fbSut(
	bExtractData:= TRUE, 
	nExtractChars:=0 , 
	sPrefix:='$01' , 
	sSuffix:= '$04', 
	bIgnoreCase:= FALSE, 
	eExtractMode := E_STRING_ExtrMode.WITHIDENT, 
	sDataString:= aDataString[1], 
	bStringFound=> , 
	sExtractedString=>, 
	nExtractedStringPos=> ,
	nExtractedStringLen=>nResult ,
	nDataStringLen=> );
	
	
	AssertEquals_UDINT(	Expected:= 83, 
						Actual:= nResult, 
						Message:= 'Extr data in mode:WITHIDENT not as expect');
				
fbSut(
	bExtractData:= TRUE, 
	nExtractChars:=0 , 
	sPrefix:='$01' , 
	sSuffix:= '$04', 
	bIgnoreCase:= FALSE, 
	eExtractMode := E_STRING_ExtrMode.WITHIDENT, 
	sDataString:= aDataString[1], 
	bStringFound=> , 
	sExtractedString=>, 
	nExtractedStringPos=> ,
	nExtractedStringLen=>nResult ,
	nDataStringLen=> );
	
	
	AssertEquals_UDINT(	Expected:= 84, 
						Actual:= nResult, 
						Message:= 'Extr data in mode:WITHIDENT not as expect');
						
fbSut(
	bExtractData:= TRUE, 
	nExtractChars:=0 , 
	sPrefix:='$01' , 
	sSuffix:= '$04', 
	bIgnoreCase:= FALSE, 
	eExtractMode := E_STRING_ExtrMode.WITHIDENT, 
	sDataString:= aDataString[1], 
	bStringFound=> , 
	sExtractedString=>, 
	nExtractedStringPos=> ,
	nExtractedStringLen=>nResult ,
	nDataStringLen=> );
	
	
	AssertEquals_UDINT(	Expected:= 82, 
						Actual:= nResult, 
						Message:= 'Extr data in mode:WITHIDENT not as expect');
						
fbSut(
	bExtractData:= TRUE, 
	nExtractChars:=0 , 
	sPrefix:='$01' , 
	sSuffix:= '$04', 
	bIgnoreCase:= FALSE, 
	eExtractMode := E_STRING_ExtrMode.WITHIDENT, 
	sDataString:= aDataString[1], 
	bStringFound=> , 
	sExtractedString=>, 
	nExtractedStringPos=> ,
	nExtractedStringLen=>nResult ,
	nDataStringLen=> );
	
	
	AssertEquals_UDINT(	Expected:= 83, 
						Actual:= nResult, 
						Message:= 'Extr data in mode:WITHIDENT not as expect');
				
TEST_FINISHED();
END_METHOD

METHOD INTERNAL testMain09_ExtractCharOnly_LeftStringWithExtractCharLenght
VAR
	fbSut 			: FB_ExtractAnyString;
	nResult 		: UDINT;	// Result
END_VAR
VAR_INST
	aDataString		: ARRAY[1..4] OF T_LongSTRING;
END_VAR
TEST('testMain09_ExtractCharOnly_LeftStringWithExtractCharLenght');	
			
aDataString[1] := '$01ST=53;$02CT=10;DS=GZDNP5JOA3IL;OG=3;XP=-50;YP=50;AP=-88;CS=06.2;SC=0070;QS=3;PN=1;$03$04$01ST=53;$02CT=10;DS=N7E1Y89UNK3O;OG=3;XP=-50;YP=-50;AP=-88;CS=06.2;SC=0070;QS=3;PN=2;$03$04'; 
					
fbSut(
	bExtractData:= TRUE, 
	nExtractChars:=82 , 
	sPrefix:='$01' , 
	sSuffix:= '$04', 
	bIgnoreCase:= FALSE, 
	eExtractMode := E_STRING_ExtrMode.WITHIDENT, 
	sDataString:= aDataString[1], 
	bStringFound=> , 
	sExtractedString=>, 
	nExtractedStringPos=> ,
	nExtractedStringLen=>nResult ,
	nDataStringLen=> );
	
	AssertEquals_STRING(Expected:= '$01ST=53;$02CT=10;DS=GZDNP5JOA3IL;OG=3;XP=-50;YP=50;AP=-88;CS=06.2;SC=0070;QS=3;PN=1;$03$04', 
						Actual:= fbSut.sExtractedString, 
						Message:= 'Extr string in mode:WITHIDENT not as expect');
						
	AssertEquals_STRING(Expected:= '$01ST=53;$02CT=10;DS=N7E1Y89UNK3O;OG=3;XP=-50;YP=-50;AP=-88;CS=06.2;SC=0070;QS=3;PN=2;$03$04', 
						Actual:= aDataString[1], 
						Message:= 'Remain string in mode:WITHIDENT not as expect');
						
	AssertEquals_UDINT(	Expected:= 83, 
						Actual:= fbSut.nExtractedStringLen, 
						Message:= 'Extr data in mode:WITHIDENT not as expect');
				
	
TEST_FINISHED();
END_METHOD

METHOD INTERNAL testNeg01_ReverseIdentAllModes_EmptyString
VAR_INST
	fbSut 			: FB_ExtractAnyString;
	aDataString		: ARRAY[1..6] OF T_LongSTRING;
	sResult 		: T_LongSTRING;	// Result
END_VAR

// '$01ST=53;$02CT=10;DS=]d201062533414058582101485MV125000156300$1D24010120957;OG=3;XP=94;YP=-39;AP=-88;CS=06.2;SC=0070;PN=1;QS=3;$03$04';
TEST('testNeg01_ReverseIdentAllModes_EmptyString');

aDataString[1] := '$01ST=53;$02CT=10;DS=]d201062533414058582101485MV125000156300$1D24010120957;OG=3;XP=94;YP=-39;AP=-88;CS=06.2;SC=0070;PN=1;QS=3;$03$04'; 
fbSut(
	bExtractData:= TRUE, 
	nExtractChars:=0 , 
	sPrefix:=';OG' , 
	sSuffix:= 'DS=', 
	bIgnoreCase:= FALSE, 
	eExtractMode := E_STRING_ExtrMode.WITHIDENT, 
	sDataString:= aDataString[1], 
	bStringFound=> , 
	sExtractedString=>sResult, 
	nExtractedStringPos=> ,
	nExtractedStringLen=> ,
	nDataStringLen=> );
	
	
	AssertEquals_STRING(	Expected:= '', 
						Actual:= sResult, 
						Message:= 'Extr data in mode:WITHIDENT not as expect');
						
	AssertEquals_STRING(	Expected:= '$01ST=53;$02CT=10;DS=]d201062533414058582101485MV125000156300$1D24010120957;OG=3;XP=94;YP=-39;AP=-88;CS=06.2;SC=0070;PN=1;QS=3;$03$04', 
						Actual:= aDataString[1], 
						Message:= 'Remaining string 1 is not as expected');
			
aDataString[2] := '$01ST=53;$02CT=10;DS=]d201062533414058582101485MV125000156300$1D24010120957;OG=3;XP=94;YP=-39;AP=-88;CS=06.2;SC=0070;PN=1;QS=3;$03$04'; 
fbSut(
	bExtractData:= TRUE, 
	nExtractChars:=0 , 
	sPrefix:=';OG' , 
	sSuffix:= 'DS=', 
	bIgnoreCase:= FALSE, 
	eExtractMode := E_STRING_ExtrMode.WITHIDENT_PURGE, 
	sDataString:= aDataString[2], 
	bStringFound=> , 
	sExtractedString=>sResult, 
	nExtractedStringPos=> ,
	nExtractedStringLen=> ,
	nDataStringLen=> );
	
	
	AssertEquals_STRING(	Expected:= '', 
						Actual:= sResult, 
						Message:= 'Extr data in mode:WITHIDENT_PURGE not as expect');
						
	AssertEquals_STRING(	Expected:= '$01ST=53;$02CT=10;DS=]d201062533414058582101485MV125000156300$1D24010120957;OG=3;XP=94;YP=-39;AP=-88;CS=06.2;SC=0070;PN=1;QS=3;$03$04', 
						Actual:= aDataString[2], 
						Message:= 'Remaining string 2 is not as expected');
						
			
aDataString[3] := '$01ST=53;$02CT=10;DS=]d201062533414058582101485MV125000156300$1D24010120957;OG=3;XP=94;YP=-39;AP=-88;CS=06.2;SC=0070;PN=1;QS=3;$03$04'; 
fbSut(
	bExtractData:= TRUE, 
	nExtractChars:=0 , 
	sPrefix:=';OG' , 
	sSuffix:= 'DS=', 
	bIgnoreCase:= FALSE, 
	eExtractMode := E_STRING_ExtrMode.WITHOUTIDENT, 
	sDataString:= aDataString[3], 
	bStringFound=> , 
	sExtractedString=>sResult, 
	nExtractedStringPos=> ,
	nExtractedStringLen=> ,
	nDataStringLen=> );
	
	
	AssertEquals_STRING(	Expected:= '', 
						Actual:= sResult, 
						Message:= 'Extr data in mode:WITHOUTIDENT not as expect');
						
	AssertEquals_STRING(	Expected:= '$01ST=53;$02CT=10;DS=]d201062533414058582101485MV125000156300$1D24010120957;OG=3;XP=94;YP=-39;AP=-88;CS=06.2;SC=0070;PN=1;QS=3;$03$04', 
						Actual:= aDataString[3], 
						Message:= 'Remaining string 3 is not as expected');
						
			
aDataString[4] := '$01ST=53;$02CT=10;DS=]d201062533414058582101485MV125000156300$1D24010120957;OG=3;XP=94;YP=-39;AP=-88;CS=06.2;SC=0070;PN=1;QS=3;$03$04'; 
fbSut(
	bExtractData:= TRUE, 
	nExtractChars:=0 , 
	sPrefix:=';OG' , 
	sSuffix:= 'DS=', 
	bIgnoreCase:= FALSE, 
	eExtractMode := E_STRING_ExtrMode.WITHOUTIDENT_PURGE, 
	sDataString:= aDataString[4], 
	bStringFound=> , 
	sExtractedString=>sResult, 
	nExtractedStringPos=> ,
	nExtractedStringLen=> ,
	nDataStringLen=> );
	
	
	AssertEquals_STRING(	Expected:= '', 
						Actual:= sResult, 
						Message:= 'Extr data in mode:WITHOUTIDENT_PURGE not as expect');
						
	AssertEquals_STRING(	Expected:= '$01ST=53;$02CT=10;DS=]d201062533414058582101485MV125000156300$1D24010120957;OG=3;XP=94;YP=-39;AP=-88;CS=06.2;SC=0070;PN=1;QS=3;$03$04', 
						Actual:= aDataString[4], 
						Message:= 'Remaining string 4 is not as expected');
						
			
aDataString[5] := '$01ST=53;$02CT=10;DS=]d201062533414058582101485MV125000156300$1D24010120957;OG=3;XP=94;YP=-39;AP=-88;CS=06.2;SC=0070;PN=1;QS=3;$03$04'; 
fbSut(
	bExtractData:= TRUE, 
	nExtractChars:=0 , 
	sPrefix:=';OG' , 
	sSuffix:= 'DS=', 
	bIgnoreCase:= FALSE, 
	eExtractMode := E_STRING_ExtrMode.WITHOUTIDENT_REMIDENT, 
	sDataString:= aDataString[5], 
	bStringFound=> , 
	sExtractedString=>sResult, 
	nExtractedStringPos=> ,
	nExtractedStringLen=> ,
	nDataStringLen=> );
	
	
	AssertEquals_STRING(	Expected:= '', 
						Actual:= sResult, 
						Message:= 'Extr data in mode:WITHOUTIDENT_REMIDENT not as expect');
						
	AssertEquals_STRING(	Expected:= '$01ST=53;$02CT=10;DS=]d201062533414058582101485MV125000156300$1D24010120957;OG=3;XP=94;YP=-39;AP=-88;CS=06.2;SC=0070;PN=1;QS=3;$03$04', 
						Actual:= aDataString[5], 
						Message:= 'Remaining string 5 is not as expected');
						
			
aDataString[6] := '$01ST=53;$02CT=10;DS=]d201062533414058582101485MV125000156300$1D24010120957;OG=3;XP=94;YP=-39;AP=-88;CS=06.2;SC=0070;PN=1;QS=3;$03$04'; 
fbSut(
	bExtractData:= TRUE, 
	nExtractChars:=0 , 
	sPrefix:=';OG' , 
	sSuffix:= 'DS=', 
	bIgnoreCase:= FALSE, 
	eExtractMode := E_STRING_ExtrMode.WITHOUTIDENT_REMIDENT_PURGE, 
	sDataString:= aDataString[6], 
	bStringFound=> , 
	sExtractedString=>sResult, 
	nExtractedStringPos=> ,
	nExtractedStringLen=> ,
	nDataStringLen=> );
	
	
	AssertEquals_STRING(	Expected:= '', 
						Actual:= sResult, 
						Message:= 'Extr data in mode:WITHOUTIDENT_REMIDENT_PURGE not as expect');
						
	AssertEquals_STRING(	Expected:= '$01ST=53;$02CT=10;DS=]d201062533414058582101485MV125000156300$1D24010120957;OG=3;XP=94;YP=-39;AP=-88;CS=06.2;SC=0070;PN=1;QS=3;$03$04', 
						Actual:= aDataString[6], 
						Message:= 'Remaining string 6 is not as expected');
				
TEST_FINISHED();
END_METHOD

METHOD INTERNAL testNeg02_NoSufixFound_EmptyStringNoDataCahnge
VAR
	fbSut 			: FB_ExtractAnyString;
	sResult			: T_LongSTRING;	// Result
	nResult 		: UDINT;	// Result
	nDataResult		: UDINT;
	
	nDataOrigin	: UDINT;
END_VAR
VAR_INST
	sDataString		: T_LongSTRING;
END_VAR
TEST('testNeg02_NoSufixFound_EmptyStringNoDataCahnge');	
			
sDataString := '$01ST=53;$02CT=10;DS=GZDNP5JOA3IL;OG=3;XP=-50;YP=50;AP=-88;CS=06.2;SC=0070;QS=3;PN=1;$03
					$01ST=53;$02CT=10;DS=N7E1Y89UNK3O;OG=3;XP=-50;YP=-50;AP=-88;CS=06.2;SC=0070;QS=3;PN=2;$03
					$01ST=53;$02CT=10;DS=JHWJXYFNX9DS;OG=3;XP=50;YP=50;AP=-88;CS=06.2;SC=0070;QS=3;PN=3;$03
					$01ST=53;$02CT=10;DS=XGBEZLBV8A9I;OG=3;XP=50;YP=-50;AP=-88;CS=06.2;SC=0070;QS=3;PN=4;$03'; 

nDataOrigin	:= len2(ADR(sDataString));
					
fbSut(
	bExtractData:= TRUE, 
	nExtractChars:=0 , 
	sPrefix:='$01' , 
	sSuffix:= '$04', 
	bIgnoreCase:= FALSE, 
	eExtractMode := E_STRING_ExtrMode.WITHIDENT, 
	sDataString:= sDataString, 
	bStringFound=> , 
	sExtractedString=>sResult, 
	nExtractedStringPos=> ,
	nExtractedStringLen=>nResult ,
	nDataStringLen=>nDataResult );
	
	AssertEquals_STRING(	Expected:= '', 
						Actual:= sResult, 
						Message:= 'Extracted string is not as expected');
						
	AssertEquals_UDINT(	Expected:= 0, 
						Actual:= nResult, 
						Message:= 'Extr data in mode:WITHIDENT not as expect');
						
	AssertEquals_UDINT(	Expected:= nDataOrigin, 
						Actual:= nDataResult, 
						Message:= 'Left data in mode:WITHIDENT not as expect');
						
TEST_FINISHED();
END_METHOD

METHOD INTERNAL testNeg03_NoPrefixFound_EmptyStringNoDataCahnge : REFERENCE TO FB_Test
VAR
	fbSut 			: FB_ExtractAnyString;
	sResult			: T_LongSTRING;	// Result
	nResult 		: UDINT;	// Result
	nDataResult		: UDINT;
	
	nDataOrigin	: UDINT;
END_VAR
VAR_INST
	sDataString		: T_LongSTRING;
END_VAR
TEST('testNeg03_NoPrefixFound_EmptyStringNoDataCahnge');	
			
sDataString := 'ST=53;$02CT=10;DS=GZDNP5JOA3IL;OG=3;XP=-50;YP=50;AP=-88;CS=06.2;SC=0070;QS=3;PN=1;$03$04
					ST=53;$02CT=10;DS=N7E1Y89UNK3O;OG=3;XP=-50;YP=-50;AP=-88;CS=06.2;SC=0070;QS=3;PN=2;$03$04
					ST=53;$02CT=10;DS=JHWJXYFNX9DS;OG=3;XP=50;YP=50;AP=-88;CS=06.2;SC=0070;QS=3;PN=3;$03$04
					ST=53;$02CT=10;DS=XGBEZLBV8A9I;OG=3;XP=50;YP=-50;AP=-88;CS=06.2;SC=0070;QS=3;PN=4;$03$04'; 

nDataOrigin	:= len2(ADR(sDataString));
					
fbSut(
	bExtractData:= TRUE, 
	nExtractChars:=0 , 
	sPrefix:='$01' , 
	sSuffix:= '$04', 
	bIgnoreCase:= FALSE, 
	eExtractMode := E_STRING_ExtrMode.WITHIDENT, 
	sDataString:= sDataString, 
	bStringFound=> , 
	sExtractedString=>sResult, 
	nExtractedStringPos=> ,
	nExtractedStringLen=>nResult ,
	nDataStringLen=>nDataResult );
	
	AssertEquals_STRING(	Expected:= '', 
						Actual:= sResult, 
						Message:= 'Extracted string is not as expected');
						
	AssertEquals_UDINT(	Expected:= 0, 
						Actual:= nResult, 
						Message:= 'Extr data in mode:WITHIDENT not as expect');
						
	AssertEquals_UDINT(	Expected:= nDataOrigin, 
						Actual:= nDataResult, 
						Message:= 'Left data in mode:WITHIDENT not as expect');
						
TEST_FINISHED();
END_METHOD

METHOD INTERNAL testNeg04_NoPrefixSufixFoundNoCharsExtr_LeftString : REFERENCE TO FB_Test
VAR
	fbSut 			: FB_ExtractAnyString;
	sResult			: T_LongSTRING;	// Result
	nResult 		: UDINT;	// Result
	nDataResult		: UDINT;
	
	nExtractedOrigin : INT;
	nDataOrigin	: UDINT;
END_VAR
VAR_INST
	sDataString		: T_LongSTRING;
END_VAR
TEST('testNeg04_NoPrefixSufixFoundNoCharsExtr_LeftString');	
			
sDataString := 'ST=53;$02CT=10;DS=GZDNP5JOA3IL;OG=3;XP=-50;YP=50;AP=-88;CS=06.2;SC=0070;QS=3;PN=1;$03$04
					ST=53;$02CT=10;DS=N7E1Y89UNK3O;OG=3;XP=-50;YP=-50;AP=-88;CS=06.2;SC=0070;QS=3;PN=2;$03$04
					ST=53;$02CT=10;DS=JHWJXYFNX9DS;OG=3;XP=50;YP=50;AP=-88;CS=06.2;SC=0070;QS=3;PN=3;$03$04
					ST=53;$02CT=10;DS=XGBEZLBV8A9I;OG=3;XP=50;YP=-50;AP=-88;CS=06.2;SC=0070;QS=3;PN=4;$03$04'; 

nExtractedOrigin := LEN('ST=53;$02CT=10;DS=GZDNP5JOA3IL;OG=3;XP=-50;YP=50;AP=-88;CS=06.2;SC=0070;QS=3;PN=1;$03$04');
nDataOrigin	:= LEN2(ADR(sDataString)) - TO_UDINT(nExtractedOrigin);
					
fbSut(
	bExtractData:= TRUE, 
	nExtractChars:=0 , 
	sPrefix:='' , 
	sSuffix:= '$04', 
	bIgnoreCase:= FALSE, 
	eExtractMode := E_STRING_ExtrMode.WITHIDENT, 
	sDataString:= sDataString, 
	bStringFound=> , 
	sExtractedString=>sResult, 
	nExtractedStringPos=> ,
	nExtractedStringLen=>nResult ,
	nDataStringLen=>nDataResult );
	
	AssertEquals_STRING( Expected:= 'ST=53;$02CT=10;DS=GZDNP5JOA3IL;OG=3;XP=-50;YP=50;AP=-88;CS=06.2;SC=0070;QS=3;PN=1;$03$04', 
						Actual:= sResult, 
						Message:= 'Extracted string is not as expected');
						
	AssertEquals_UDINT(	Expected:= TO_UDINT(nExtractedOrigin), 
						Actual:= nResult, 
						Message:= 'Extr data in mode:WITHIDENT not as expect');
						
	AssertEquals_UDINT(	Expected:= nDataOrigin, 
						Actual:= nDataResult, 
						Message:= 'Left data in mode:WITHIDENT not as expect');
						
TEST_FINISHED();
END_METHOD

METHOD INTERNAL testNeg05_PrefixFoundNoSufixNoCharsExtr_RightString : REFERENCE TO FB_Test
VAR
	fbSut 			: FB_ExtractAnyString;
	sResult			: T_LongSTRING;	// Result
	nResult 		: UDINT;	// Result
	nDataResult		: UDINT;
	
	nExtractedOrigin : UDINT;
END_VAR
VAR_INST
	sDataString		: T_LongSTRING;
END_VAR
TEST('testNeg05_PrefixFoundNoSufixNoCharsExtr_RightString');	
			
sDataString := 'ST=53;$02CT=10;DS=GZDNP5JOA3IL;OG=3;XP=-50;YP=50;AP=-88;CS=06.2;SC=0070;QS=3;PN=1;$03$04ST=53;$02CT=10;DS=N7E1Y89UNK3O;OG=3;XP=-50;YP=-50;AP=-88;CS=06.2;SC=0070;QS=3;PN=2;$03$04
					$01ST=53;$02CT=10;DS=JHWJXYFNX9DS;OG=3;XP=50;YP=50;AP=-88;CS=06.2;SC=0070;QS=3;PN=3;$03$04ST=53;$02CT=10;DS=XGBEZLBV8A9I;OG=3;XP=50;YP=-50;AP=-88;CS=06.2;SC=0070;QS=3;PN=4;$03$04'; 

nExtractedOrigin := LEN2(ADR('$01ST=53;$02CT=10;DS=JHWJXYFNX9DS;OG=3;XP=50;YP=50;AP=-88;CS=06.2;SC=0070;QS=3;PN=3;$03$04ST=53;$02CT=10;DS=XGBEZLBV8A9I;OG=3;XP=50;YP=-50;AP=-88;CS=06.2;SC=0070;QS=3;PN=4;$03$04'));
					
fbSut(
	bExtractData:= TRUE, 
	nExtractChars:=0 , 
	sPrefix:='$01' , 
	sSuffix:= '', 
	bIgnoreCase:= FALSE, 
	eExtractMode := E_STRING_ExtrMode.WITHIDENT_PURGE, 
	sDataString:= sDataString, 
	bStringFound=> , 
	sExtractedString=>sResult, 
	nExtractedStringPos=> ,
	nExtractedStringLen=>nResult ,
	nDataStringLen=>nDataResult );
	
	AssertEquals_STRING( Expected:= '$01ST=53;$02CT=10;DS=JHWJXYFNX9DS;OG=3;XP=50;YP=50;AP=-88;CS=06.2;SC=0070;QS=3;PN=3;$03$04ST=53;$02CT=10;DS=XGBEZLBV8A9I;OG=3;XP=50;YP=-50;AP=-88;CS=06.2;SC=0070;QS=3;PN=4;$03$04', 
						Actual:= sResult, 
						Message:= 'Extracted string is not as expected');
						
	AssertEquals_UDINT(	Expected:= TO_UDINT(nExtractedOrigin), 
						Actual:= nResult, 
						Message:= 'Extr data in mode:WITHIDENT_PURGE not as expect');
						
	AssertEquals_UDINT(	Expected:= 0, 
						Actual:= nDataResult, 
						Message:= 'Left data in mode:WITHIDENT_PURGE not as expect');
						
TEST_FINISHED();
END_METHOD

METHOD INTERNAL testSeq01_MVxDecode_ImageData
VAR
	fbSut01 			: FB_ExtractAnyString;
	fbSut02 			: FB_ExtractAnyString;
	fbSut03 			: FB_ExtractAnyString;
	aResult				: ARRAY[1..3] OF T_LongSTRING;	// Result
	nResult 			: UDINT;	// Result
	nDataResult			: UDINT;
	nIndex				: INT;
	nExtractedOrigin 	: UDINT;
END_VAR				
VAR_INST
	sDataString		: T_LongSTRING;		//'ST=53;$02CT=10;DS=GZDNP5JOA3IL;OG=3;XP=-50;YP=50;AP=-88;CS=06.2;SC=0070;QS=3;PN=1;$03'
	stImageData		: ST_SCANNER_ImageData;
END_VAR
TEST('testSeq01_MVxDecode_ImageData');

sDataString := 'ST=53;$02CT=10;DS=GZDNP5JOA3IL;OG=3;XP=-50;YP=50;AP=-88;CS=06.2;SC=0070;QS=3;PN=1;$03'; 

	(* get image data message *)
	//fbCodeData
	fbSut01(
		nExtractChars:=0 , 
		sPrefix:='$02' , 
		sSuffix:= '$03', 
		bIgnoreCase:= FALSE, 
		eExtractMode := E_STRING_ExtrMode.WITHOUTIDENT_REMIDENT, 
		sDataString:= sDataString, 
		bStringFound=> , 
		sExtractedString=>aResult[1], 
		nExtractedStringPos=> ,
		nExtractedStringLen=> ,
		nDataStringLen=> );
	
		AssertEquals_STRING( Expected:= 'ST=53;', 
						Actual:= sDataString, 
						Message:= 'Extr data in mode:WITHOUTIDENT_REMIDENT not as expect');
						
		AssertEquals_STRING( Expected:= 'CT=10;DS=GZDNP5JOA3IL;OG=3;XP=-50;YP=50;AP=-88;CS=06.2;SC=0070;QS=3;PN=1;', 
						Actual:= aResult[1], 
						Message:= 'Extr data in mode:WITHOUTIDENT_REMIDENT not as expect');

	(* code data found *)
	IF fbSut01.bStringFound THEN
		
		nIndex := 1;
		
		//fbFieldData
		fbSut02(
			nExtractChars:=0 , 
			sPrefix:='CT=' , 
			sSuffix:= ';', 
			bIgnoreCase:= FALSE, 
			eExtractMode := E_STRING_ExtrMode.WITHOUTIDENT_REMIDENT_PURGE, 
			sDataString:= fbSut01.sExtractedString, 
			bStringFound=> , 
			sExtractedString=>, 
			nExtractedStringPos=> ,
			nExtractedStringLen=> ,
			nDataStringLen=> );
			
		IF fbSut02.bStringFound THEN
			(* extract data value *)
			stImageData.aCodeData[nIndex].eCodeType := STRING_TO_INT(fbSut02.sExtractedString);
		END_IF
		
		AssertEquals_INT(	Expected:= E_SCANNER_CodeType.DATAMARTIX,
					Actual:= stImageData.aCodeData[nIndex].eCodeType, 
					Message:= 'Extr data in mode:WITHOUTIDENT_REMIDENT_PURGE not as expect');
						
		fbSut02(
			nExtractChars:=0 , 
			sPrefix:='DS=' , 
			sSuffix:= ';OG=', 
			bIgnoreCase:= FALSE, 
			eExtractMode := E_STRING_ExtrMode.WITHOUTIDENT_PURGE, 
			sDataString:= fbSut01.sExtractedString, 
			bStringFound=> , 
			sExtractedString=>aResult[2], 
			nExtractedStringPos=> ,
			nExtractedStringLen=> ,
			nDataStringLen=> );
		
		IF fbSut02.bStringFound THEN
			(* extract data value *)
			stImageData.aCodeData[nIndex].strDataString := fbSut02.sExtractedString;
		END_IF
		
		AssertEquals_STRING( Expected:= 'GZDNP5JOA3IL', 
				Actual:= aResult[2], 
				Message:= 'Extr data in mode:WITHOUTIDENT_PURGE not as expect');
		
		IF LEN(stImageData.aCodeData[nIndex].strDataString) > 0 AND stImageData.aCodeData[nIndex].eCodeType <> E_SCANNER_CodeType.NONE THEN
			
			fbSut03(
				nExtractChars:=0 , 
				sPrefix:='OG=' , 
				sSuffix:= ';', 
				bIgnoreCase:= FALSE, 
				eExtractMode := E_STRING_ExtrMode.WITHOUTIDENT_REMIDENT, 
				sDataString:= fbSut01.sExtractedString, 
				bStringFound=> , 
				sExtractedString=>, 
				nExtractedStringPos=> ,
				nExtractedStringLen=> ,
				nDataStringLen=> );
			
			IF fbSut03.bStringFound THEN
				(* extract data value *)
				stImageData.aCodeData[nIndex].fOverallGrade := STRING_TO_LREAL(fbSut03.sExtractedString);
			END_IF
			
			AssertEquals_LREAL(Expected:= 3, 
						Actual:= stImageData.aCodeData[nIndex].fOverallGrade, 
						Delta:= 0.001, 
						Message:= 'Extr data in mode:WITHOUTIDENT_REMIDENT not as expect' );
			
			fbSut03(
				nExtractChars:=0 , 
				sPrefix:='QS=' , 
				sSuffix:= ';', 
				bIgnoreCase:= FALSE, 
				eExtractMode := E_STRING_ExtrMode.WITHOUTIDENT_REMIDENT, 
				sDataString:= fbSut01.sExtractedString, 
				bStringFound=> , 
				sExtractedString=>, 
				nExtractedStringPos=> ,
				nExtractedStringLen=> ,
				nDataStringLen=> );
			
			IF fbSut03.bStringFound THEN
				(* extract data value *)
				stImageData.aCodeData[nIndex].nEvaluation := STRING_TO_INT(fbSut03.sExtractedString);
			END_IF
									
			AssertEquals_INT(	Expected:= 3, 
						Actual:= stImageData.aCodeData[nIndex].nEvaluation, 
						Message:= 'Left data in mode:WITHIDENT_PURGE not as expect');
			
			fbSut03(
				nExtractChars:=0 , 
				sPrefix:='YP=' , 		//XP and YP reversed intetnionally to check if alghoritm is resistant for change order
				sSuffix:= ';', 
				bIgnoreCase:= FALSE, 
				eExtractMode := E_STRING_ExtrMode.WITHOUTIDENT_REMIDENT, 
				sDataString:= fbSut01.sExtractedString, 
				bStringFound=> , 
				sExtractedString=>, 
				nExtractedStringPos=> ,
				nExtractedStringLen=> ,
				nDataStringLen=> );
			
			IF fbSut03.bStringFound THEN
				(* extract data value *)
				stImageData.aCodeData[nIndex].fYPos := STRING_TO_LREAL(fbSut03.sExtractedString);
			END_IF
			
			AssertEquals_LREAL(Expected:= 50, 
				Actual:= stImageData.aCodeData[nIndex].fYPos, 
				Delta:= 0.001, 
				Message:= 'Extr data in mode:WITHOUTIDENT_REMIDENT not as expect' );
	
			fbSut03(
				nExtractChars:=0 , 
				sPrefix:='XP=' , 
				sSuffix:= ';', 
				bIgnoreCase:= FALSE, 
				eExtractMode := E_STRING_ExtrMode.WITHOUTIDENT_REMIDENT, 
				sDataString:= fbSut01.sExtractedString, 
				bStringFound=> , 
				sExtractedString=>, 
				nExtractedStringPos=> ,
				nExtractedStringLen=> ,
				nDataStringLen=> );
			
			IF fbSut03.bStringFound THEN
				(* extract data value *)
				stImageData.aCodeData[nIndex].fXPos := STRING_TO_LREAL(fbSut03.sExtractedString);
			END_IF
			
			AssertEquals_LREAL(Expected:= -50, 
				Actual:= stImageData.aCodeData[nIndex].fXPos, 
				Delta:= 0.001, 
				Message:= 'Extr data in mode:WITHOUTIDENT_REMIDENT not as expect' );
				
			fbSut03(
				nExtractChars:=0 , 
				sPrefix:='CS=' , 
				sSuffix:= ';', 
				bIgnoreCase:= FALSE, 
				eExtractMode := E_STRING_ExtrMode.WITHOUTIDENT_REMIDENT, 
				sDataString:= fbSut01.sExtractedString, 
				bStringFound=> , 
				sExtractedString=>, 
				nExtractedStringPos=> ,
				nExtractedStringLen=> ,
				nDataStringLen=> );
			
			IF fbSut03.bStringFound THEN
				(* extract data value *)
				stImageData.aCodeData[nIndex].fCellSize := STRING_TO_LREAL(fbSut03.sExtractedString);
			END_IF
			
			AssertEquals_LREAL(Expected:= 6.2, 
				Actual:= stImageData.aCodeData[nIndex].fCellSize, 
				Delta:= 0.001, 
				Message:= 'Extr data in mode:WITHOUTIDENT_REMIDENT not as expect' );
				
			fbSut03(
				nExtractChars:=0 , 
				sPrefix:='SC=' , 
				sSuffix:= ';', 
				bIgnoreCase:= FALSE, 
				eExtractMode := E_STRING_ExtrMode.WITHOUTIDENT_REMIDENT, 
				sDataString:= fbSut01.sExtractedString, 
				bStringFound=> , 
				sExtractedString=>, 
				nExtractedStringPos=> ,
				nExtractedStringLen=> ,
				nDataStringLen=> );
			
			IF fbSut03.bStringFound THEN
				(* extract data value *)
				stImageData.aCodeData[nIndex].fSymbolContrast := STRING_TO_LREAL(fbSut03.sExtractedString);
			END_IF
			
			AssertEquals_LREAL(Expected:= 70, 
				Actual:= stImageData.aCodeData[nIndex].fSymbolContrast, 
				Delta:= 0.001, 
				Message:= 'Extr data in mode:WITHOUTIDENT_REMIDENT not as expect' );
		END_IF
		
		fbSut02(
			nExtractChars:=0 , 
			sPrefix:='PN=' , 
			sSuffix:= ';', 
			bIgnoreCase:= FALSE, 
			eExtractMode := E_STRING_ExtrMode.WITHOUTIDENT_REMIDENT_PURGE, 
			sDataString:= fbSut01.sExtractedString, 
			bStringFound=> , 
			sExtractedString=>, 
			nExtractedStringPos=> ,
			nExtractedStringLen=> ,
			nDataStringLen=> nResult);
		
		IF fbSut02.bStringFound THEN
			(* extract data value *)
			stImageData.aCodeData[nIndex].nProgramNo := STRING_TO_BYTE(fbSut02.sExtractedString);
		END_IF
		
		AssertEquals_BYTE(	Expected:= 1, 
						Actual:= stImageData.aCodeData[nIndex].nProgramNo, 
						Message:= 'Extr data in mode:WITHOUTIDENT_REMIDENT_PURGE not as expect');
						
	END_IF
	
	
	AssertEquals_STRING( Expected:= '',
						Actual:= fbSut01.sExtractedString,
						Message:= 'Extracted string is not as expected');
						
	AssertEquals_UDINT(	Expected:= 0, 
						Actual:= nResult, 
						Message:= 'Extr data in mode:WITHIDENT_PURGE not as expect');

//Check no additional string

	fbSut01(
		nExtractChars:=0 , 
		sPrefix:='$02' , 
		sSuffix:= '$03', 
		bIgnoreCase:= FALSE, 
		eExtractMode := E_STRING_ExtrMode.WITHOUTIDENT_REMIDENT, 
		sDataString:= sDataString, 
		bStringFound=> , 
		sExtractedString=>, 
		nExtractedStringPos=> ,
		nExtractedStringLen=>nDataResult ,
		nDataStringLen=> );
	
	AssertEquals_UDINT( Expected:= 0, 
						Actual:= fbSut01.nExtractedStringLen, 
						Message:= 'Extr data in mode:WITHOUTIDENT_REMIDENT not as expect');
						
	(* code data found *)
	IF NOT fbSut01.bStringFound AND nIndex = 1 THEN					
		
		stImageData.nCodesRead	:= nIndex;
		(* Scan Time field (ST=%c;) *)
		fbSut02(
			nExtractChars:=0 , 
			sPrefix:='ST=' , 
			sSuffix:= ';', 
			bIgnoreCase:= FALSE, 
			eExtractMode := E_STRING_ExtrMode.WITHOUTIDENT_REMIDENT_PURGE, 
			sDataString:= sDataString, 
			bStringFound=> , 
			sExtractedString=>aResult[3], 
			nExtractedStringPos=> ,
			nExtractedStringLen=> nDataResult,
			nDataStringLen=> );
			
		IF fbSut02.bStringFound THEN
			(* extract data value *)
			stImageData.tScanTime := UDINT_TO_TIME(STRING_TO_UDINT(fbSut02.sExtractedString));
		END_IF
	END_IF
		
	AssertEquals_STRING( Expected:= '', 
					Actual:= sDataString, 
					Message:= 'Extr data in mode:WITHOUTIDENT_REMIDENT_PURGE not as expect');
					
	AssertEquals_TIME( Expected:= T#53MS, 
					Actual:= stImageData.tScanTime, 
					Message:= 'Extr data in mode:WITHOUTIDENT_REMIDENT_PURGE not as expect');

	
	TEST_FINISHED();
END_METHOD

END_FUNCTION_BLOCK

// ---- POUs/METS/Common LIB/08_SOFTWARE LIB/String FBs/FB_ExtractAnyString.TcPOU
// Extracts a sub-string defined by prefix and suffix 
// Works in one cycle but as FB to not use stack memore due to LongString data defined
FUNCTION_BLOCK FB_ExtractAnyString
VAR_INPUT
	bExtractData			: BOOL;			(* set TRUE to remove prefix and suffix from strData *)
	nExtractChars			: UDINT;			(* if suffix is blank, number of data chars to extract *)
	sPrefix					: T_LongSTRING;	(* prefix string extended from T_MaxString to T_LongSTRING *)
	sSuffix					: T_LongSTRING;	(* suffix string extended from T_MaxString to T_LongSTRING *)
	bIgnoreCase				: BOOL;
	eExtractMode			: E_STRING_ExtrMode	:= E_STRING_ExtrMode.WITHOUTIDENT_REMIDENT;
	//bIncludeIdentifiers	: BOOL;
END_VAR
VAR_IN_OUT
	sDataString				: T_LongSTRING;	(* string to be searched *)
END_VAR
VAR_OUTPUT
	bStringFound			: BOOL;			(* TRUE = sub-string with matching prefix/suffix found *)
	sExtractedString		: T_LongSTRING;	(* extracted data *)
	nExtractedStringPos		: UDINT;			(* start pos of extracted string in strString *)
	nExtractedStringLen		: UDINT;
	nDataStringLen			: UDINT;
END_VAR
VAR
	
	//_rtExecute			: R_trig;
	
	_nExtractChars			: UDINT;
	_sPrefix				: T_LongSTRING;	(* prefix string *)
	_sSuffix				: T_LongSTRING;	(* suffix string *)
	_sDataString			: T_LongSTRING;	(* string to be searched *)
	
	_bIncludeIdentifiers	: BOOL;
	_bPurgeFullString		: BOOL;
	
	_nDataStringLen			: UDINT;
	_nPrefixLen				: UDINT;
	_nSuffixLen				: UDINT;
	
	_bPrefixFound			: BOOL;
	_bSuffixFound			: BOOL;
	
	_bPrefixIndex			: UDINT;
	_bTempSuffixIndex		: UDINT;
	_bSuffixIndex			: UDINT;
	
	_nStartDataPos			: UDINT;
	_nAbsolutDataPos		: UDINT;
	_nEndDataPos			: UDINT;
	_nExtractedDataLen		: UDINT;
	
	_nTerminatePos			: UDINT;
END_VAR

//	EXTRWITHIDENT						//extract with ident and dont purge left side string
//	EXTRWITHIDENT_PURGE					//extract with ident and purge left side string
//	EXTRWITHOUTIDENT					//extract with ident and dont purge left side string, both ident left in origin string 
//	EXTRWITHOUTIDENT_PURGE				//extract with ident and purge left side string, only sufix ident left in origin string
//	EXTRWITHOUTIDENT_REMIDENT			//extract with ident and dont purge left side string, no ident left in origin string
//	EXTRWITHOUTIDENT_REMIDENT_PURGE		//extract with ident and purge left side string, no ident left in origin string

//====================================================================================	
IF 	eExtractMode = E_STRING_ExtrMode.WITHIDENT 			OR 
	eExtractMode = E_STRING_ExtrMode.WITHIDENT_PURGE 	THEN
	
	_bIncludeIdentifiers	:= TRUE;
ELSE 
	_bIncludeIdentifiers	:= FALSE;
END_IF

IF 	eExtractMode = E_STRING_ExtrMode.WITHIDENT_PURGE 		OR 
	eExtractMode = E_STRING_ExtrMode.WITHOUTIDENT_PURGE 	OR 
	eExtractMode = E_STRING_ExtrMode.WITHOUTIDENT_REMIDENT_PURGE THEN
	
	_bPurgeFullString	:= LEN2(ADR(sDataString)) = SIZEOF(sDataString)-1;
ELSE 
	_bPurgeFullString	:= FALSE;
END_IF

//====================================================================================	

(* rising edge of bExecute *)
//_rtExecute(CLK := bExtractData);

//IF _rtExecute.Q THEN
	
//====================================================================================	
	bStringFound 		:= FALSE;
	
	_sDataString 		:= '';
	_sPrefix 			:= '';
	_sSuffix 			:= '';
	
	_bPrefixFound		:= FALSE;
	_bSuffixFound		:= FALSE;
		
	_bPrefixIndex		:= 0;
	_bSuffixIndex		:= 0;
		
	_nStartDataPos		:= 0;
	_nAbsolutDataPos	:= 0;
	_nEndDataPos		:= 0;
	//_ExtractedDataLen	:= 0;
	
	 (*calc string lengths *)
	_nDataStringLen 	:= LEN2(ADR(sDataString));
	_nPrefixLen 		:= LEN2(ADR(sPrefix));
	_nSuffixLen 		:= LEN2(ADR(sSuffix));
	
	_nExtractChars:= LIMIT(0, nExtractChars, _nDataStringLen);
	
	(*clear outputs*)
	nExtractedStringPos	:= 0;
	nExtractedStringLen	:= 0;
	nDataStringLen		:= _nDataStringLen;

//====================================================================================	
	
	(* matching for Prefix and Suffix is case-sesnsitive - worsk only with T_MaxString *)
	IF bIgnoreCase AND 
		_nDataStringLen < 256 	AND 
		_nPrefixLen < 256 		AND 
		_nSuffixLen < 256 		THEN
		
		(* internal comparators are all converted to lower case *)
		_sDataString 	:= F_ToLCase(sDataString);
		_sPrefix 		:= F_ToLCase(sPrefix);
		_sSuffix 		:= F_ToLCase(sSuffix);
		
	ELSE
		(* internal comparators are not changed *)
		_sDataString 	:= sDataString;
		_sPrefix 		:= sPrefix;
		_sSuffix 		:= sSuffix;
	END_IF

//====================================================================================	

	IF _nPrefixLen = 0 AND  _nExtractChars > 0 THEN
		
		_bPrefixIndex		:= 1;
		_nStartDataPos		:= 1;
		nExtractedStringPos := 1;
		
	ELSIF _nPrefixLen > 0 THEN		//if _nPrefixLen = 0 then _bPrefixIndex and _StartDataPos remains 0 from init state
		
		_bPrefixIndex	:= FIND2(ADR(_sDataString), ADR(_sPrefix));		//find search only if prefix declared on the input
	
		IF _bPrefixIndex > 0 THEN		//_bPrefixIndex as result form find can be onlu positive range
			
			_bPrefixFound := TRUE;		// _bPrefixFound guarantee _StartDataPos > 0
			_nStartDataPos 	:= SEL(_bIncludeIdentifiers, _bPrefixIndex + _nPrefixLen, _bPrefixIndex);
			_nAbsolutDataPos	:= _bPrefixIndex + _nPrefixLen;
			
			nExtractedStringPos := _nStartDataPos;
		END_IF
	END_IF	
	
//====================================================================================		

	IF _nSuffixLen = 0 AND  _nExtractChars > 0 THEN //IF only nExtractChars is declared THEN _EndDataPos pointing on elemnt determinated by nExtractChars or on last elemnt OF DataString
		
		_bSuffixIndex := _bPrefixIndex + _nPrefixLen + _nExtractChars;
		_nEndDataPos := MIN(_bSuffixIndex, _nDataStringLen);
		
		IF _nEndDataPos > _nStartDataPos THEN  // check if both pointers not point on last DataString elemnt
			_bSuffixFound := TRUE;	// _bSuffixFound guarantee _EndDataPos > 0 and found after _StartDataPos
		END_IF
		
	ELSIF _nSuffixLen > 0 THEN // if _nSuffixLen declared, then ignor nExtractChars and search for find sufix position using 
		
		// Include Sufix change shift if onle Prfix was found >> SEL(_bPrefixFound, 0, _StartDataPos - 1)
		_bTempSuffixIndex	:= FIND2(ADR(_sDataString) + SEL(_bPrefixFound, 0, _nAbsolutDataPos - 1), ADR(_sSuffix)); //find search only if sufix declared on the input and on index after prefix
		IF _bTempSuffixIndex > 0 THEN
			_bSuffixIndex	:= _bTempSuffixIndex + SEL(_bPrefixFound, 0, _nAbsolutDataPos - 1);	//Recalculate Sufix real position if sufix found or _bSuffixIndex remain 0 form init
		END_IF
		
		(*_bTempSuffixIndex gurantee that sufix was search after prefix position so _EndDataPos always greater than _StartDataPos *) 
		IF _bSuffixIndex > 0 THEN
			_bSuffixFound := TRUE;	// _bSuffixFound guarantee _EndDataPos > 0
			_nEndDataPos := SEL(_bIncludeIdentifiers,_bSuffixIndex, _bSuffixIndex + _nSuffixLen);
		END_IF
	END_IF
	
//====================================================================================		
	
	MEMSET(ADR(sExtractedString), 16#00, SIZEOF(sExtractedString));	//Clean sExtractedString area for new data

	IF _bPrefixFound AND _bSuffixFound THEN

		DELETE2(ADR(sDataString), ADR(sExtractedString), SIZEOF(sExtractedString), 
											SIZEOF(sExtractedString) - _nEndDataPos , _nEndDataPos);
		DELETE2(ADR(sExtractedString), ADR(sExtractedString), SIZEOF(sExtractedString), _nStartDataPos -1, 1);
		
	ELSIF _nPrefixLen = 0 AND _nSuffixLen = 0 AND _nExtractChars >= _nEndDataPos THEN		
		
		sExtractedString := sDataString;
		
	ELSIF _nPrefixLen = 0 AND _bSuffixFound THEN		// TO BE CONSIDERED IF WE WANT THIS CONDITION - IT WORKS LIKE LEFT
		
		_nStartDataPos := 1;
		DELETE2(ADR(sDataString), ADR(sExtractedString), SIZEOF(sExtractedString), 
										SIZEOF(sExtractedString) - _nEndDataPos , _nEndDataPos);
										
	ELSIF _bPrefixFound AND _nSuffixLen = 0 AND _nExtractChars = 0 THEN
		
		_nEndDataPos		:= _nDataStringLen;
		DELETE2(ADR(sDataString), ADR(sExtractedString), SIZEOF(sExtractedString), _nStartDataPos -1, 1);
		
	END_IF
		
	nExtractedStringLen	:= LEN2(ADR(sExtractedString));
	IF nExtractedStringLen <> 0 THEN  bStringFound := TRUE; END_IF
	
//====================================================================================
	IF NOT bStringFound AND _bPurgeFullString THEN
		
		sDataString := '';
		nDataStringLen := 0;
		
	ELSIF sExtractedString = sDataString THEN
		
		sDataString := '';
		nDataStringLen := 0;
		
	ELSIF bStringFound THEN //Terminate DataString only if endpositin for sufix is determinated and guratnee _EndDataPos greater then 0
		
		CASE eExtractMode OF

			E_STRING_ExtrMode.WITHIDENT:
			
				DELETE2(ADR(sDataString), ADR(sDataString), SIZEOF(sDataString), nExtractedStringLen, _nStartDataPos);		
					
			E_STRING_ExtrMode.WITHIDENT_PURGE:	
			
				IF _nEndDataPos = _nDataStringLen THEN
					DELETE2(ADR(sDataString), ADR(sDataString), SIZEOF(sDataString), _nEndDataPos, 1);
				ELSE
					DELETE2(ADR(sDataString), ADR(sDataString), SIZEOF(sDataString), _nEndDataPos -1, 1);
				END_IF
					
			E_STRING_ExtrMode.WITHOUTIDENT:		
			
				 DELETE2(ADR(sDataString), ADR(sDataString), SIZEOF(sDataString), nExtractedStringLen, _nStartDataPos);	
		
			E_STRING_ExtrMode.WITHOUTIDENT_PURGE:
						
				IF _nEndDataPos = _nDataStringLen THEN
					DELETE2(ADR(sDataString), ADR(sDataString), SIZEOF(sDataString), _nEndDataPos, 1);
				ELSE
					DELETE2(ADR(sDataString), ADR(sDataString), SIZEOF(sDataString), _nEndDataPos -1, 1);
				END_IF
				
			E_STRING_ExtrMode.WITHOUTIDENT_REMIDENT:
			
				DELETE2(ADR(sDataString), ADR(sDataString), SIZEOF(sDataString), 
										nExtractedStringLen + _nPrefixLen + _nSuffixLen, _bPrefixIndex);	
		
			E_STRING_ExtrMode.WITHOUTIDENT_REMIDENT_PURGE:		
						
				IF _nEndDataPos = _nDataStringLen THEN
					DELETE2(ADR(sDataString), ADR(sDataString), SIZEOF(sDataString), _nEndDataPos, 1);
				ELSE
					DELETE2(ADR(sDataString), ADR(sDataString), SIZEOF(sDataString), _bSuffixIndex + _nSuffixLen -1, 1);
				END_IF
				
		ELSE
			
			DELETE2(ADR(sDataString), ADR(sDataString), SIZEOF(sDataString), 
							nExtractedStringLen + _nPrefixLen + _nSuffixLen, _bPrefixIndex);
							
		END_CASE
	
		nDataStringLen := LEN2(ADR(sDataString));
	END_IF
//END_IF


(*

		
		IF _bSuffixIndex > _nDataStringLen THEN	//_EndDataPos cannot bi greater then _nDataStringLen due to previuse min condition
			_ExtractedDataLen := _EndDataPos -_StartDataPos + 1; // if _EndDataPos pointing on last element of sDataString, we must include it ofr extratcion
		ELSE
			_ExtractedDataLen := _EndDataPos -_StartDataPos;	//if prefix and sufix are found  _ExtractedDataLen always greater than 0
		END_IF
		
		MEMMOVE(ADR(sExtractedString),ADR(sDataString) + _StartDataPos -1 , _ExtractedDataLen);	// _StartDataPos -1 as initial adress has alredy value 1
		//MEMSET(ADR(sExtractedString) + _ExtractedDataLen, 16#00, _nDataStringLen - _ExtractedDataLen);
		
		
		
		//MEMMOVE(ADR(sExtractedString),ADR(sDataString), _EndDataPos);
		//MEMSET(ADR(sExtractedString) + _EndDataPos, 16#00, _nDataStringLen - _EndDataPos);
		
		
		
	
		IF _bSuffixIndex > _nDataStringLen THEN	//_EndDataPos cannot bi greater then _nDataStringLen due to previuse min condition
			_nTerminatePos := _EndDataPos;
		ELSE
			_nTerminatePos := SEL(_bIncludeIdentifiers, _EndDataPos + _nSuffixLen, _EndDataPos) -1; //sub 1 from final result as adressing of char start form pos 1
			//so if Terminate index should be 10 then _nTerminatePos must be 9 to add with initial addres of DataString
		END_IF
		
		IF _nDataStringLen > _nTerminatePos THEN	// guarantee we are not operating beyond DataString area
			MEMMOVE(ADR(sDataString), ADR(sDataString) + _nTerminatePos, _nDataStringLen - _nTerminatePos);
			MEMSET(ADR(sDataString) + _nDataStringLen - _nTerminatePos, 16#00, _nTerminatePos);
		ELSIF _nDataStringLen <= _nTerminatePos THEN
			sDataString := '';
		END_IF
			
	*)

END_FUNCTION_BLOCK

// ---- POUs/TcUnit/FB_ExtractStringTests/FB_ExtratcStringTests.TcPOU
FUNCTION_BLOCK FB_ExtratcStringTests EXTENDS FB_TestSuite

//==============================================================
//MAIN TESTS
//==============================================================

//fbExtracStringTests_bExtractDataSetFalse_ExtractedDSWtihExtraChar();
//fbExtracStringTests_bExtractDataSetFalse_ExtractedDSAndOGWtihExtraChar();

//fbExtracStringTests_bExtractDataSetTrue_ExtractedDSWtihoutExtraChar();
//fbExtracStringTests_bExtractDataSetTrue_ExtractedDSAndOGWtihoutExtraChar();

METHOD INTERNAL fbExtracStringTests_bExtractDataSetFalse_ExtractedDSAndOGWtihExtraChar
VAR
	fbSut		: FB_ExtractString;
	
	sDataString	: T_MaxString	:= '$01ST=53;$02CT=10;DS=]d201062533414058582101485MV125000165300$1D24010120957;OG=3;XP=94;YP=-39;AP=-88;CS=06.2;SC=0070;PN=1;QS=3;$03$04';	(* string to be searched *)
END_VAR
// At FB_SCANNER_MVxDecodeImageData
TEST('fbExtracStringTests_bExtractDataSetFalse_ExtractedDSAndOGWtihExtraChar');

fbSut(
	bExtractData:= FALSE , 
	nExtractChars:=0 , 
	strPrefix:= 'DS=', 
	strSuffix:= ';OG=', 
	strString:= sDataString , 
	bStringFound=> , 
	nStartPos=> , 
	strData=> );
	
	AssertEquals_STRING(	Expected:= 'DS=]d201062533414058582101485MV125000165300$1D24010120957;OG=' , 
					Actual:= fbSut.strData, 
					Message:= 'Extracted string is not as expected');
					
	fbSut(
	bExtractData:= FALSE , 
	nExtractChars:=0 , 
	strPrefix:= 'OG=', 
	strSuffix:= ';', 
	strString:= sDataString , 
	bStringFound=> , 
	nStartPos=> , 
	strData=> );


	AssertEquals_STRING(	Expected:= 'OG=3;' , 
						Actual:= fbSut.strData, 
						Message:= 'Extracted string is not as expected');
	
						
TEST_FINISHED();
END_METHOD

METHOD INTERNAL fbExtracStringTests_bExtractDataSetFalse_ExtractedDSWtihExtraChar
VAR
	fbSut		: FB_ExtractString;
	
	sDataString	: T_MaxString	:= '$01ST=53;$02CT=10;DS=]d201062533414058582101485MV125000165300$1D24010120957;OG=3;XP=94;YP=-39;AP=-88;CS=06.2;SC=0070;PN=1;QS=3;$03$04';	(* string to be searched *)
END_VAR
// At FB_SCANNER_MVxDecodeImageData
TEST('fbExtracStringTests_bExtractDataSetFalse_ExtractedDSWtihExtraChar');

fbSut(
	bExtractData:= FALSE , 
	nExtractChars:=0 , 
	strPrefix:= 'DS=', 
	strSuffix:= ';OG=', 
	strString:= sDataString , 
	bStringFound=> , 
	nStartPos=> , 
	strData=> );


	AssertEquals_STRING(	Expected:= 'DS=]d201062533414058582101485MV125000165300$1D24010120957;OG=' , 
						Actual:= fbSut.strData, 
						Message:= 'Extracted string is not as expected');
						
	AssertEquals_STRING(	Expected:= '$01ST=53;$02CT=10;3;XP=94;YP=-39;AP=-88;CS=06.2;SC=0070;PN=1;QS=3;$03$04', 
						Actual:= sDataString, 
						Message:= 'Remaining string is not as expected');
						
TEST_FINISHED();
END_METHOD

METHOD INTERNAL fbExtracStringTests_bExtractDataSetTrue_ExtractedDSAndOGWtihoutExtraChar
VAR
	fbSut		: FB_ExtractString;
	
	sDataString	: T_MaxString	:= '$01ST=53;$02CT=10;DS=]d201062533414058582101485MV125000165300$1D24010120957;OG=3;XP=94;YP=-39;AP=-88;CS=06.2;SC=0070;PN=1;QS=3;$03$04';	(* string to be searched *)
END_VAR
// At FB_SCANNER_MVxDecodeImageData
//
//Input string: '$01ST=53;$02CT=10;DS=]d201062533414058582101485MV125000165300$1D24010120957;OG=3;XP=94;YP=-39;AP=-88;CS=06.2;SC=0070;PN=1;QS=3;$03$04'
//
//		fbFieldData(
//			bExtractData	:= TRUE,
//			strPrefix		:= 'DS=',
//			strSuffix		:= ';OG=',
//			strString		:= fbCodeData.strData
//		);
//(* Overall Grade field (OG=%Q0;) *)
//			fbFieldData(
//				bExtractData	:= TRUE,
//				strPrefix		:= 'OG=',
//				strSuffix		:= ';',
//				strString		:= fbCodeData.strData
//			);


TEST('fbExtracStringTests_bExtractDataSetTrue_ExtractedDSAndOGWtihoutExtraChar');

fbSut(
	bExtractData:= TRUE , 
	nExtractChars:=0 , 
	strPrefix:= 'DS=', 
	strSuffix:= ';OG=', 
	strString:= sDataString , 
	bStringFound=> , 
	nStartPos=> , 
	strData=> );
	
	AssertEquals_STRING(	Expected:= ']d201062533414058582101485MV125000165300$1D24010120957' , 
					Actual:= fbSut.strData, 
					Message:= 'Extracted string is not as expected');
						
	fbSut(
	bExtractData:= TRUE , 
	nExtractChars:=0 , 
	strPrefix:= 'OG=', 
	strSuffix:= ';', 
	strString:= sDataString , 
	bStringFound=> , 
	nStartPos=> , 
	strData=> );


	AssertEquals_STRING(	Expected:= '3' , 
						Actual:= fbSut.strData, 
						Message:= 'Extracted string is not as expected');
						
						
TEST_FINISHED();
END_METHOD

METHOD INTERNAL fbExtracStringTests_bExtractDataSetTrue_ExtractedDSWtihoutExtraChar
VAR
	fbSut		: FB_ExtractString;
	
	sDataString	: T_MaxString	:= '$01ST=53;$02CT=10;DS=]d201062533414058582101485MV125000165300$1D24010120957;OG=3;XP=94;YP=-39;AP=-88;CS=06.2;SC=0070;PN=1;QS=3;$03$04';	(* string to be searched *)
END_VAR
// At FB_SCANNER_MVxDecodeImageData
//
//Input string: '$01ST=53;$02CT=10;DS=]d201062533414058582101485MV125000165300$1D24010120957;OG=3;XP=94;YP=-39;AP=-88;CS=06.2;SC=0070;PN=1;QS=3;$03$04'
//
//		fbFieldData(
//			bExtractData	:= TRUE,
//			strPrefix		:= 'DS=',
//			strSuffix		:= ';OG=',
//			strString		:= fbCodeData.strData
//		);

TEST('fbExtracStringTests_bExtractDataSetTrue_ExtractedDSWtihoutExtraChar');

fbSut(
	bExtractData:= TRUE , 
	nExtractChars:=0 , 
	strPrefix:= 'DS=', 
	strSuffix:= ';OG=', 
	strString:= sDataString , 
	bStringFound=> , 
	nStartPos=> , 
	strData=> );


	AssertEquals_STRING(	Expected:= ']d201062533414058582101485MV125000165300$1D24010120957' , 
						Actual:= fbSut.strData, 
						Message:= 'Extracted string is not as expected');
						
	AssertEquals_STRING(	Expected:= '$01ST=53;$02CT=10;3;XP=94;YP=-39;AP=-88;CS=06.2;SC=0070;PN=1;QS=3;$03$04', 
						Actual:= sDataString, 
						Message:= 'Remaining string is not as expected');
						
TEST_FINISHED();
END_METHOD

END_FUNCTION_BLOCK

// ---- POUs/METS/Common LIB/08_SOFTWARE LIB/String FBs/FB_ExtractString.TcPOU
(* extracts a sub-string defined by prefix and suffix *)
FUNCTION_BLOCK FB_ExtractString
VAR_INPUT
	bExtractData		: BOOL;			(* set TRUE to remove prefix and suffix from strData *)
	nExtractChars		: UINT;			(* if suffix is blank, number of data chars to extract *)
	strPrefix			: T_MaxString;	(* prefix string *)
	strSuffix			: T_MaxString;	(* suffix string *)
END_VAR
VAR_IN_OUT
	strString			: T_MaxString;	(* string to be searched *)
END_VAR
VAR_OUTPUT
	bStringFound		: BOOL;			(* TRUE = sub-string with matching prefix/suffix found *)
	nStartPos			: UINT;			(* start pos of extracted string in strString *)
	strData				: T_MaxString;	(* extracted data *)
END_VAR
VAR
	nStringLen			: UINT;
	nPrefixLen			: UINT;
	nSuffixLen			: UINT;
	nEndPos				: UINT;
	bStartPosFound		: BOOL;
	bEndPosFound		: BOOL;
	nChars				: UINT;
	nMaxIndex			: UINT;
	nIndex				: UINT;
END_VAR
(*
-------------------------------------------------------------------------------------------------
DATE		Version	Author	Comments
-------------------------------------------------------------------------------------------------
30/01/2015	3.00.00	PB		bExtractData input added to specify whether prefix and suffix should be removed from strData
							bIgnoreCase input removed
							Major optimisation to reduce time taken to find a string

-------------------------------------------------------------------------------------------------
06/09/2012	1.41.00	PB		strData output added which returns strResult without the prefix and suffix
06/07/2011	1.23.00	PB		Pre-check added to ensure that strString is not empty
07/06/2011	1.19.00	PB		bIgnoreCase input added, set to TRUE to ignore upper/lower case when matching Prefix and Suffix
31/01/2011	1.08.03	PB		Bug fix - strings now handled correctly if strSuffix is longer than 1 char
							Search for suffix changed to start after prefix position
22/11/2010	1.07.01	PB		Initial release

-------------------------------------------------------------------------------------------------
*)

(* calc string lengths *)
nStringLen := INT_TO_UINT(LEN(strString));
nPrefixLen := INT_TO_UINT(LEN(strPrefix));
nSuffixLen := INT_TO_UINT(LEN(strSuffix));

(* string to be searched is not empty and prefix or suffix or no or chars to extract is defined *)
IF nStringLen > 0 AND (nPrefixLen > 0 OR nSuffixLen > 0 OR nExtractChars > 0) THEN

	(* clear outputs *)
	bStringFound := FALSE;
	nChars := 0;
	nStartPos := 0;
	strData := '';

	(* initialise char index values *)
	bStartPosFound := FALSE;
	bEndPosFound := FALSE;
	nEndPos := 0;

	(* max search index, based on string length - 1 due to starting at 0 and length of prefix *)
	nMaxIndex := (nStringLen - 1) + (nPrefixLen - 1);

	(* for each character in the string *)
	FOR nIndex := 0 TO nMaxIndex DO

		(* prefix has not been found *)
		IF bStartPosFound = FALSE THEN

			(* no prefix defined  *)
			IF nPrefixLen = 0 THEN

				(* start at beginning if string *)
				nStartPos := 1;
				bStartPosFound := TRUE;

			(* prefix defined  *)
			ELSE

				(* compare partial string with prefix *)
				IF MEMCMP(ADR(strString) + nIndex, ADR(strPrefix), nPrefixLen) = 0 THEN

					(* prefix position found *)
					nStartPos := nIndex + 1;
					bStartPosFound := TRUE;

					(* skip to end of prefix to continue search *)
					nIndex := nIndex + nPrefixLen - 1;
				END_IF
			END_IF

		(* suffix has not been found *)
		ELSIF bEndPosFound = FALSE THEN

			(* no suffix defined  *)
			IF nSuffixLen = 0 THEN

				(* start at 1st char of string *)
				bEndPosFound := TRUE;

				(* calculate end position *)
				nEndPos := MIN((nStartPos - 1) + nExtractChars + nPrefixLen, nStringLen);

			(* suffix defined  *)
			ELSE

				(* compare partial string with suffix *)
				IF MEMCMP(ADR(strString) + nIndex, ADR(strSuffix), nSuffixLen) = 0 THEN

					(* suffix position found, calculate end position *)
					nEndPos := nIndex + nSuffixLen;
					bEndPosFound := TRUE;

					(* no prefix defined and number of chars to extract is defined *)
					IF nPrefixLen = 0 AND nExtractChars > 0 THEN

						(* re-calculate start position *)
						nStartPos := MAX(nEndPos - nExtractChars - 1, 1);
					END_IF

					(* search complete, quit FOR loop *)
					EXIT;
				END_IF
			END_IF

		(* prefix and suffix found *)
		ELSE

			(* quit FOR loop *)
			EXIT;
		END_IF
	END_FOR

	(* start and end positions known *)
	IF bStartPosFound = TRUE AND bEndPosFound = TRUE THEN

		(* string has been found *)
		bStringFound := TRUE;

		(* return string without prefix and suffix *)
		IF bExtractData = TRUE THEN

			(* total chars to be moved to strData *)
			nChars := (nEndPos - (nStartPos - 1)) - nPrefixLen - nSuffixLen;

			(* 1 or more chars to be moved *)
			IF nChars > 0 THEN

				(* move data to strData *)
				MEMMOVE(ADR(strData), ADR(strString) + (nStartPos - 1) + nPrefixLen, nChars);
			END_IF

		(* return string with prefix and suffix *)
		ELSE

			(* total chars to be moved to strData *)
			nChars := nEndPos - (nStartPos - 1);

			(* 1 or more chars to be moved *)
			IF nChars > 0 THEN

				(* move data to strData *)
				MEMMOVE(ADR(strData), ADR(strString) + (nStartPos - 1), nChars);
			END_IF
		END_IF

		(* terminate strData *)
		MEMSET(ADR(strData) + nChars, 16#00, 1);

		(* 1 or more chars after strSuffix *)
		IF nStringLen > (nEndPos - (nStartPos - 1)) THEN

			(* shift post-suffix chars to prefix position *)
			MEMMOVE(ADR(strString) + (nStartPos - 1), ADR(strString) + nEndPos, nStringLen - (nEndPos - (nStartPos - 1)));
		END_IF

		(* terminate strString *)
		MEMSET(ADR(strString) + nStringLen - (nEndPos - (nStartPos - 1)), 16#00, 1);
	END_IF

(* string to be searched is empty or prefix and suffix and both blank *)
ELSE

	(* clear outputs *)
	bStringFound := FALSE;
	nChars := 0;
	strData := '';
END_IF

END_FUNCTION_BLOCK

// ---- POUs/TcUnit/FUN_ReplaceLongSingleCharTests/FB_ReplaceLongStringCharTests.TcPOU
FUNCTION_BLOCK FB_ReplaceLongStringCharTests EXTENDS FB_TestSuite

//==============================================================
//MAIN TESTS
//==============================================================

testMain01_ExtractCharFromLongString_AllCahrsExtracted();
testMain02_RepalceCharFromLongString_AllCahrsRepalced();

//==============================================================
//NEGATIVE TESTS
//==============================================================

testNeg01_ReplaceInputs_NoChangeInFullCode();
testNeg02_TwoCharsOnInputs_OneCharReplaced();

//==============================================================
//SEQUENCE TESTS
//==============================================================

//==============================================================
//OTHERS TESTS
//==============================================================

METHOD INTERNAL testMain01_ExtractCharFromLongString_AllCahrsExtracted
VAR
	
	sFullCode			: T_LongSTRING;	
	sExpectedResult		: T_LongSTRING;
	sActualResult		: T_LongSTRING;
END_VAR
TEST('testMain01_ExtractCharFromLongString_AllCahrsExtracted');

sFullCode := 'ST=53;$02CT=10;DS=GZDNP5JOA3IL$1D;OG=3;XP=-50;YP=50;AP=-88;CS=06.2;SC=0070;QS=3;PN=1;$03$04
											ST=53;$02CT=10;DS=N7E1Y89UNK3O$1D;OG=3;XP=-50;YP=-50;AP=-88;CS=06.2;SC=0070;QS=3;PN=2;$03$04
											ST=53;$02CT=10;DS=JHWJXYFNX9DS$1D;OG=3;XP=50;YP=50;AP=-88;CS=06.2;SC=0070;QS=3;PN=3;$03$04
											ST=53;$02CT=10;DS=XGBEZLBV8A9I$1D;OG=3;XP=50;YP=-50;AP=-88;CS=06.2;SC=0070;QS=3;PN=4;$03$04'; 

sExpectedResult := 'ST=53;$02CT=10;DS=GZDNP5JOA3IL;OG=3;XP=-50;YP=50;AP=-88;CS=06.2;SC=0070;QS=3;PN=1;$03$04
											ST=53;$02CT=10;DS=N7E1Y89UNK3O;OG=3;XP=-50;YP=-50;AP=-88;CS=06.2;SC=0070;QS=3;PN=2;$03$04
											ST=53;$02CT=10;DS=JHWJXYFNX9DS;OG=3;XP=50;YP=50;AP=-88;CS=06.2;SC=0070;QS=3;PN=3;$03$04
											ST=53;$02CT=10;DS=XGBEZLBV8A9I;OG=3;XP=50;YP=-50;AP=-88;CS=06.2;SC=0070;QS=3;PN=4;$03$04'; 


sActualResult	:= F_ReplaceLongSingleChar(sFullCode:= sFullCode, 
							sCharRemove:= '$1D', 
							sReplacmentChar:='' );
							
AssertEquals_STRING(Expected:= sExpectedResult, 
						Actual:= sActualResult, 
						Message:= 'Extracted string is not as expected');
						
TEST_FINISHED();
END_METHOD

METHOD INTERNAL testMain02_RepalceCharFromLongString_AllCahrsRepalced
VAR
	
	sFullCode			: T_LongSTRING;	
	sExpectedResult		: T_LongSTRING;
	sActualResult		: T_LongSTRING;
END_VAR
TEST('testMain02_RepalceCharFromLongString_AllCahrsRepalced');

sFullCode := 'ST=53;$02CT=10;DS=GZDNP5JOA3IL$1D;OG=3;XP=-50;YP=50;AP=-88;CS=06.2;SC=0070;QS=3;PN=1;$03$04
											ST=53;$02CT=10;DS=N7E1Y89UNK3O$1D;OG=3;XP=-50;YP=-50;AP=-88;CS=06.2;SC=0070;QS=3;PN=2;$03$04
											ST=53;$02CT=10;DS=JHWJXYFNX9DS$1D;OG=3;XP=50;YP=50;AP=-88;CS=06.2;SC=0070;QS=3;PN=3;$03$04
											ST=53;$02CT=10;DS=XGBEZLBV8A9I$1D;OG=3;XP=50;YP=-50;AP=-88;CS=06.2;SC=0070;QS=3;PN=4;$03$04'; 

sExpectedResult := 'ST=53;$02CT=10;DS=GZDNP5JAA3IL$1D;AG=3;XP=-50;YP=50;AP=-88;CS=06.2;SC=0070;QS=3;PN=1;$03$04
											ST=53;$02CT=10;DS=N7E1Y89UNK3A$1D;AG=3;XP=-50;YP=-50;AP=-88;CS=06.2;SC=0070;QS=3;PN=2;$03$04
											ST=53;$02CT=10;DS=JHWJXYFNX9DS$1D;AG=3;XP=50;YP=50;AP=-88;CS=06.2;SC=0070;QS=3;PN=3;$03$04
											ST=53;$02CT=10;DS=XGBEZLBV8A9I$1D;AG=3;XP=50;YP=-50;AP=-88;CS=06.2;SC=0070;QS=3;PN=4;$03$04'; 


sActualResult	:= F_ReplaceLongSingleChar(sFullCode:= sFullCode, 
							sCharRemove:= 'O', 
							sReplacmentChar:='A' );
							
AssertEquals_STRING(Expected:= sExpectedResult, 
						Actual:= sActualResult, 
						Message:= 'Extracted string is not as expected');
						
TEST_FINISHED();
END_METHOD

METHOD INTERNAL testNeg01_ReplaceInputs_NoChangeInFullCode
VAR
	
	sFullCode			: T_LongSTRING;	
	sExpectedResult		: T_LongSTRING;
	sActualResult		: T_LongSTRING;
END_VAR
TEST('testNeg01_ReplaceInputs_NoChangeInFullCode');

sFullCode := 'ST=53;$02CT=10;DS=GZDNP5JOA3IL$1D;OG=3;XP=-50;YP=50;AP=-88;CS=06.2;SC=0070;QS=3;PN=1;$03$04
											ST=53;$02CT=10;DS=N7E1Y89UNK3O$1D;OG=3;XP=-50;YP=-50;AP=-88;CS=06.2;SC=0070;QS=3;PN=2;$03$04
											ST=53;$02CT=10;DS=JHWJXYFNX9DS$1D;OG=3;XP=50;YP=50;AP=-88;CS=06.2;SC=0070;QS=3;PN=3;$03$04
											ST=53;$02CT=10;DS=XGBEZLBV8A9I$1D;OG=3;XP=50;YP=-50;AP=-88;CS=06.2;SC=0070;QS=3;PN=4;$03$04'; 

sExpectedResult := 'ST=53;$02CT=10;DS=GZDNP5JOA3IL$1D;OG=3;XP=-50;YP=50;AP=-88;CS=06.2;SC=0070;QS=3;PN=1;$03$04
											ST=53;$02CT=10;DS=N7E1Y89UNK3O$1D;OG=3;XP=-50;YP=-50;AP=-88;CS=06.2;SC=0070;QS=3;PN=2;$03$04
											ST=53;$02CT=10;DS=JHWJXYFNX9DS$1D;OG=3;XP=50;YP=50;AP=-88;CS=06.2;SC=0070;QS=3;PN=3;$03$04
											ST=53;$02CT=10;DS=XGBEZLBV8A9I$1D;OG=3;XP=50;YP=-50;AP=-88;CS=06.2;SC=0070;QS=3;PN=4;$03$04'; 


sActualResult	:= F_ReplaceLongSingleChar(sFullCode:= sFullCode, 
							sCharRemove:= '', 
							sReplacmentChar:='$1D' );
							
AssertEquals_STRING(Expected:= sExpectedResult, 
						Actual:= sActualResult, 
						Message:= 'Extracted string is not as expected');
						
TEST_FINISHED();
END_METHOD

METHOD INTERNAL testNeg02_TwoCharsOnInputs_OneCharReplaced
VAR
	
	sFullCode			: T_LongSTRING;	
	sExpectedResult		: T_LongSTRING;
	sActualResult		: T_LongSTRING;
END_VAR
TEST('testNeg02_TwoCharsOnInputs_OneCharReplaced');

sFullCode := 'ST=53;$02CT=10;DS=GZDNP5JOA3IL$1D;OG=3;XP=-50;YP=50;AP=-88;CS=06.2;SC=0070;QS=3;PN=1;$03$04
											ST=53;$02CT=10;DS=N7E1Y89UNK3O$1D;OG=3;XP=-50;YP=-50;AP=-88;CS=06.2;SC=0070;QS=3;PN=2;$03$04
											ST=53;$02CT=10;DS=JHWJXYFNX9DS$1D;OG=3;XP=50;YP=50;AP=-88;CS=06.2;SC=0070;QS=3;PN=3;$03$04
											ST=53;$02CT=10;DS=XGBEZLBV8A9I$1D;OG=3;XP=50;YP=-50;AP=-88;CS=06.2;SC=0070;QS=3;PN=4;$03$04'; 

sExpectedResult := 'ST=53;$02CT=10;DS=GZDNP5JOA3IL$1D;OG=3;XP=-50;YP=50;AP=-88;CS=06.2;SC=0070;QS=3;PN=1;$1D$04
											ST=53;$02CT=10;DS=N7E1Y89UNK3O$1D;OG=3;XP=-50;YP=-50;AP=-88;CS=06.2;SC=0070;QS=3;PN=2;$1D$04
											ST=53;$02CT=10;DS=JHWJXYFNX9DS$1D;OG=3;XP=50;YP=50;AP=-88;CS=06.2;SC=0070;QS=3;PN=3;$1D$04
											ST=53;$02CT=10;DS=XGBEZLBV8A9I$1D;OG=3;XP=50;YP=-50;AP=-88;CS=06.2;SC=0070;QS=3;PN=4;$1D$04';


{warning disable C0198}

sActualResult	:= F_ReplaceLongSingleChar(sFullCode:= sFullCode, 
							sCharRemove:= '$03$04', 
							sReplacmentChar:='$1D' );
{warning restore C0198}	
						
AssertEquals_STRING(Expected:= sExpectedResult, 
						Actual:= sActualResult, 
						Message:= 'Extracted string is not as expected');
						
TEST_FINISHED();
END_METHOD

END_FUNCTION_BLOCK

// ---- POUs/METS/Common LIB/08_SOFTWARE LIB/String FBs/F_ReplaceLongSingleChar.TcPOU
FUNCTION F_ReplaceLongSingleChar : T_LongSTRING
VAR_INPUT
	sFullCode		: T_LongSTRING;
	sCharRemove			: T_Char := '$1D';
	sReplacmentChar		: T_Char := '';
END_VAR
VAR
	sCodeSize		: STRING;
END_VAR

WHILE FIND2(ADR(sFullCode), ADR(sCharRemove)) > 0 DO
	REPLACE2(ADR(sFullCode),ADR(sReplacmentChar), ADR(sFullCode), 
						SIZEOF(sFullCode), LEN2(ADR(sCharRemove)), FIND2(ADR(sFullCode), ADR(sCharRemove)));
END_WHILE

(*Diagnostic part for long stirng operation *)
//sCodeSize := TO_STRING(LEN2(ADR(sFullCode)));
//CONCAT2(ADR(sCodeSize), ADR('_'), ADR(sCodeSize), SIZEOF(sCodeSize));	
//INSERT2(ADR(sFullCode), ADR(sCodeSize), ADR(sFullCode), SIZEOF(sFullCode), 0);
	
F_ReplaceLongSingleChar	:= sFullCode;

END_FUNCTION

// ---- POUs/TcUnit/FB_LOGHandlerTests/FB_LogHandlerTests.TcPOU
FUNCTION_BLOCK FB_LogHandlerTests EXTENDS FB_TestSuite

//==============================================================
//MAIN TESTS
//==============================================================

testMain01_ReducedMaxImageSize_BufferOverflow();

//==============================================================
//NEGATIVE TESTS
//==============================================================

//==============================================================
//SEQUENCE TESTS
//==============================================================

//==============================================================
//OTHERS TESTS
//==============================================================

METHOD INTERNAL testMain01_ReducedMaxImageSize_BufferOverflow
VAR
	fbLogHandler			: FB_LOG_Handler;
	sLogMessage				: T_LongSTRING;
	
END_VAR
VAR_INST
	stEventDataUT				: ST_LOG_EventData;
END_VAR
TEST('testMain01_ReducedMaxImageSize_BufferOverflow');

stEventDataUT.bEnable := TRUE;
//stEventDataUT.sTimeStamp :=MID( F_SYSTEM_SystemTimeAsISO8601(gDevice.stMetsStatus.stCTDateTime.sSystemTime, gDevice.stMetsStatus.stCTDateTime.sUTCTimeZoneOffset ), 12, 12);
stEventDataUT.nMaxImageArraySize	:= 300;
sLogMessage := '$01ST=53;$02CT=10;DS=GZDNP5JOA3IL;OG=3;XP=-50;YP=50;AP=-88;CS=06.2;SC=0070;QS=3;PN=1;$03
					$01ST=53;$02CT=10;DS=N7E1Y89UNK3O;OG=3;XP=-50;YP=-50;AP=-88;CS=06.2;SC=0070;QS=3;PN=2;$03
					$01ST=53;$02CT=10;DS=JHWJXYFNX9DS;OG=3;XP=50;YP=50;AP=-88;CS=06.2;SC=0070;QS=3;PN=3;$03
					$01ST=53;$02CT=10;DS=XGBEZLBV8A9I;OG=3;XP=50;YP=-50;AP=-88;CS=06.2;SC=0070;QS=3;PN=4;$03';


fbLogHandler(
	_IsUsed:= TRUE, 
	bLogData:= TRUE , 
	sLogMessage:= sLogMessage , 
	stEventData:= stEventDataUT, 
	bDone=> , 
	bBufferOverflow=> );


AssertEquals_BOOL(Expected := TRUE, 
						Actual:= fbLogHandler.bBufferOverflow, 
						Message:= 'Buffer output state not as expected');
					
TEST_FINISHED();
END_METHOD

END_FUNCTION_BLOCK

// ---- POUs/METS/Common LIB/08_SOFTWARE LIB/Logger FBs/FB_LOG_Handler.TcPOU
FUNCTION_BLOCK FB_LOG_Handler
VAR_INPUT
	_IsUsed					: BOOL;
	bLogData					: BOOL;
	sLogMessage				: T_LongSTRING;
END_VAR
VAR_IN_OUT
	stEventData				: ST_LOG_EventData;
END_VAR
VAR_OUTPUT
	bDone						: BOOL;
	bBufferOverflow			: BOOL;
END_VAR
VAR
	rtExecute					: R_TRIG;
	sString 					: T_LongSTRING;
	nStringLen					: UINT;

END_VAR

_IsUsed := TRUE;

rtExecute(CLK:=bLogData);

IF NOT stEventData.bBufferOverflow AND stEventData.bEnable AND sLogMessage <> '' AND rtExecute.Q THEN

	sString := '';
	(*stEventData.nCounter := stEventData.nCounter + 1;
	sString := F_CONCAT4(F_AddPaddingUDINT(stEventData.nCounter, 7), ' : ', stEventData.sTimeStamp, ' : ');*)
	//sString := CONCAT(stEventData.sTimeStamp, ' : ');
	//sString := F_LongCONCAT(sString,sLogMessage);
	//sString := F_LongCONCAT(sString,'.$R$N');
	CONCAT2(ADR(stEventData.sTimeStamp), ADR(' : '), ADR(sString), SIZEOF(sString));
	CONCAT2(ADR(sString), ADR(sLogMessage), ADR(sString), SIZEOF(sString));
	CONCAT2(ADR(sString), ADR('.$R$N'), ADR(sString), SIZEOF(sString));
	nStringLen := TO_UINT(LEN2(ADR(sString)));  //Max size 1024 byte -> LongString

	stEventData.nControlSize := stEventData.nControlSize + nStringLen;

	IF stEventData.nControlSize <  stEventData.nMaxImageArraySize THEN
		MEMMOVE(ADR(stEventData.aDataLogImage[stEventData.nImageByte]), ADR(sString), nStringLen);
		stEventData.nImageByte := stEventData.nImageByte + nStringLen;
	ELSE
		stEventData.bBufferOverflow	:=TRUE;
		bBufferOverflow	:= TRUE;
	END_IF

	bDone	:= TRUE;
	(*F_LOG_Handler := TRUE;*)
ELSE
	bDone	:= FALSE;
END_IF

END_FUNCTION_BLOCK

// ---- POUs/TcUnit/FB_CASE_ValidateContentTests/FB_CASE_ValidateContentTests.TcPOU
FUNCTION_BLOCK FB_CASE_ValidateContentTests EXTENDS TcUnit.FB_TestSuite

VAR
	
(* General data *)
	stCTDateTime_tests					: ST_SYSTEM_DateTime;	
	stProductInstruction_tests			: ST_PCM_Status;
	nSecquentionalCounter_tests			: UDINT;
	stCodeInfo_Outer_tests				: ST_CodeInfo;
	stCaseRejectReasons_tests			: ST_RejectReasonsForCase;
	stRejectReasonsForOuter_tests		: ST_RejectReasonsForOuter;
	stOuterDataNotFound_tests			: ST_RejectItems;

(* 01.Main tests container *)

	stProductInstruction_test_0101		: ST_PCM_Status;
	stCACData_test_0101 				: ST_CAC_Data;
		
	stCACData_tests 					: ST_CAC_Data;
(* 02.DataConsistancy tests container *)
	stProductInstruction_test_0201		: ST_PCM_Status;
	stCACData_test_0201 				: ST_CAC_Data;
	sRejectCode_test_0201				: T_MaxString;
	
	stProductInstruction_test_0202		: ST_PCM_Status;
	stCACData_test_0202 				: ST_CAC_Data;
	sRejectCode_test_0202				: T_MaxString;	
	
	
	stProductInstruction_test_0203		: ST_PCM_Status;
	stCACData_test_0203 				: ST_CAC_Data;
	sRejectCode_test_0203				: T_MaxString;
	
	stProductInstruction_test_0204		: ST_PCM_Status;
	stCACData_test_0204 				: ST_CAC_Data;
	sRejectCode_test_0204				: T_MaxString;

	
	stProductInstruction_test_0205		: ST_PCM_Status;
	stCACData_test_0205 				: ST_CAC_Data;
	sRejectCode_test_0205				: T_MaxString;
	
	stProductInstruction_test_0206		: ST_PCM_Status;
	stCACData_test_0206 				: ST_CAC_Data;
	sRejectCode_test_0206				: T_MaxString;

(* 03.NumberOfOuters tests container *)
	stProductInstruction_test_0301		: ST_PCM_Status;
	stCACData_test_0301 				: ST_CAC_Data;
	sRejectCode_test_0301				: T_MaxString;
	
	stProductInstruction_test_0302		: ST_PCM_Status;
	stCACData_test_0302 				: ST_CAC_Data;
	sRejectCode_test_0302				: T_MaxString;
	
	stProductInstruction_test_0303		: ST_PCM_Status;
	stCACData_test_0303 				: ST_CAC_Data;
	sRejectCode_test_0303				: T_MaxString;
	
(* 04.OuterAggrDissable tests container *)
	stProductInstruction_test_0401		: ST_PCM_Status;
	stCACData_test_0401 				: ST_CAC_Data;
	sRejectCode_test_0401				: T_MaxString;
	
	stProductInstruction_test_0402		: ST_PCM_Status;
	stCACData_test_0402 				: ST_CAC_Data;
	sRejectCode_test_0402				: T_MaxString;

(* 05.OuterAggrEnable tests container *)
	stProductInstruction_test_0501		: ST_PCM_Status;
	stCACData_test_0501 				: ST_CAC_Data;
	sRejectCode_test_0501				: T_MaxString;
	
	stProductInstruction_test_0502		: ST_PCM_Status;
	stCACData_test_0502 				: ST_CAC_Data;
	sRejectCode_test_0502				: T_MaxString;

(* 06.DuplicateHandler tests container *)
	
	stProductInstruction_test_0601		: ST_PCM_Status;
	stCACData_test_0601 				: ST_CAC_Data;
	sRejectCode_test_0601				: T_MaxString;
	
	stCACData_test_0602 				: ST_CAC_Data;
	stProductInstruction_test_0602		: ST_PCM_Status;
	sRejectCode_test_0602				: T_MaxString;
	
(* 07.OACmissing tests container *)
	
	stProductInstruction_test_0701		: ST_PCM_Status;
	stCACData_test_0701 				: ST_CAC_Data;
	sRejectCode_test_0701				: T_MaxString;
	
	stCACData_test_0702 				: ST_CAC_Data;
	stProductInstruction_test_0702		: ST_PCM_Status;
	sRejectCode_test_0702				: T_MaxString;
	
	sRejectCode_tets					: T_MaxString;
	
END_VAR


//==============================================================
//01.Main
//==============================================================
main01_bExecuteFalseNoAction();
//==============================================================
//02.DataConsistancy
//==============================================================
dataConsistancy01_NumOfOutersWrong();
dataConsistancy02_NumOfOutersExceedcMAX_Outers();
dataConsistancy03_ValidationCodeNotFoundInInfeedQueue();
dataConsistancy04_OuterCodeVal_IndexErrorFound();
dataConsistancy05_NumberOfOutersToSmall();
dataConsistancy06_NumberOfOutersToBig();

//==============================================================
//03.NumberOfOuters
//==============================================================
numberOfOuters01_ValueToLittlebErrorTrue();
numberOfOuters02_ValueGraterErrorTrue();
numberOfOuters03_ValueToLittlebErrorTrueRejectCodeWright();

//==============================================================
//04.OuterAggrDissable
//==============================================================
outerAggrDissable01_sRejectCodeOK();

//==============================================================
//05.OuterAggrEnable
//==============================================================
outerAggrEnable01_PacksPerOuterZero();
outerAggrEnable02_PacksPerCaseZero();


//==============================================================
//06.DuplicatesHandler
//==============================================================
duplicateHandler01_OuterDuplicatebErrorTrue();
duplicateHandler02_PackDuplicatebErrorTrue();

//==============================================================
//07.OACmissing
//==============================================================
oacMissing01nErrorID21();

METHOD INTERNAL dataConsistancy01_NumOfOutersWrong
VAR
	//fbCaseTest			: FB_CASE_ValidateContent;
	bDone				: BOOL;
	bBusy				: BOOL;
	bError				: BOOL;
	nErrorID 			: UDINT;
	nValidationIndex	: INT;
	
	eLastState			: E_CAC_State;
			
END_VAR

VAR_INST
	fbCaseTest0201				: FB_CASE_ValidateContent;
	rTrig0201					: R_TRIG;
	nCycles0201					: INT;
	
END_VAR

//Data initialization
TestInit(stCACData:= stCACData_test_0201, stProductInstruction:= stProductInstruction_test_0201);

//Change some data for test scenario below
stCACData_test_0201.NumberOfOuters := stCACData_test_0201.NumberOfOuters - 2;
	
TcUnit.TEST('dataConsistancy01_NumOfOutersWrong');


fbCaseTest0201(
	bExecute:= TRUE, 
	bIsDuplicateOuters:= FALSE, 
	bIsDuplicatePacks:= FALSE, 
	stCTDateTime:= stCTDateTime_tests, 
	stOuterDataNotFound:= stRejectReasonsForOuter_tests.stOuterDataNotFound, 
	stProductInstruction:= stProductInstruction_test_0201, 
	nSecquentionalCounter:= nSecquentionalCounter_tests, 
	stCodeInfo_Outer:= stCodeInfo_Outer_tests, 
	stCaseRejectReasons:= stCaseRejectReasons_tests, 
	stCACData:= stCACData_test_0201, 
	bDone=> bDone, 
	bBusy=> bBusy, 
	bError=> bError, 
	nErrorID=> nErrorID, 
	sRejectCode=> sRejectCode_test_0201, 
	nValidationIndex=> nValidationIndex
);
	
rTrig0201(CLK:= fbCaseTest0201.bDone);
nCycles0201 := nCycles0201 + 1;	

IF rTrig0201.Q THEN	
		
	AssertEquals_BOOL(Expected 	:= TRUE,
					  Actual 	:= bError,
					  Message 	:= 'Wrong number of outers not detected'
	);
	
	AssertEquals_STRING(Expected := 'XXVAL048XX',
						Actual := TO_STRING(fbCaseTest0201.sRejectCode),
						Message := 'Wrong value of nErrorID'
	);
	
	TEST_FINISHED();
	
ELSIF nCycles0201 > 50 THEN
	
	AssertTrue(Condition := TRUE,
			   Message 	 := 'Timeout dataConsistancy01_NumOfOutersWrong'
	);	 
	TEST_FINISHED();
END_IF
END_METHOD

METHOD INTERNAL dataConsistancy02_NumOfOutersExceedcMAX_Outers
VAR
	//fbCaseTest			: FB_CASE_ValidateContent;
	bDone				: BOOL;
	bBusy				: BOOL;
	bError				: BOOL;
	nErrorID 			: UDINT;
	nValidationIndex	: INT;
	
	eLastState			: E_CAC_State;
			
END_VAR

VAR_INST
	fbCaseTest0202				: FB_CASE_ValidateContent;
	rTrig0202					: R_TRIG;
	nCycles0202					: INT;
	
END_VAR

//Data initialization
TestInit(stCACData:= stCACData_test_0202, stProductInstruction:= stProductInstruction_test_0202);

//Change some data for test scenario below
stCACData_test_0202.NumberOfOuters := - 1;
	
TcUnit.TEST('dataConsistancy02_NumOfOutersExceedcMAX_Outers');


fbCaseTest0202(
	bExecute:= TRUE, 
	bIsDuplicateOuters:= FALSE, 
	bIsDuplicatePacks:= FALSE, 
	stCTDateTime:= stCTDateTime_tests, 
	stOuterDataNotFound:= stRejectReasonsForOuter_tests.stOuterDataNotFound, 
	stProductInstruction:= stProductInstruction_test_0202, 
	nSecquentionalCounter:= nSecquentionalCounter_tests, 
	stCodeInfo_Outer:= stCodeInfo_Outer_tests, 
	stCaseRejectReasons:= stCaseRejectReasons_tests, 
	stCACData:= stCACData_test_0202, 
	bDone=> bDone, 
	bBusy=> bBusy, 
	bError=> bError, 
	nErrorID=> nErrorID, 
	sRejectCode=> sRejectCode_test_0202, 
	nValidationIndex=> nValidationIndex
);
	
rTrig0202(CLK:= fbCaseTest0202.bDone);
nCycles0202 := nCycles0202 + 1;	

IF rTrig0202.Q THEN	
		
	AssertEquals_UDINT(Expected := 11,
                   	   Actual 	:= fbCaseTest0202.nErrorID,
                   	   Message 	:= 'nErrorID value wrong');
	
	TEST_FINISHED();
	
ELSIF nCycles0202 > 50 THEN
	
	AssertTrue(Condition := TRUE,
			   Message 	 := 'Timeout dataConsistancy02_NumOfOutersExceedcMAX_Outers'
	);	 
	TEST_FINISHED();
END_IF
END_METHOD

METHOD INTERNAL dataConsistancy03_ValidationCodeNotFoundInInfeedQueue
VAR
	//fbCaseTest			: FB_CASE_ValidateContent;
	bDone				: BOOL;
	bBusy				: BOOL;
	bError				: BOOL;
	nErrorID 			: UDINT;
	nValidationIndex	: INT;
	
	eLastState			: E_CAC_State;
			
END_VAR

VAR_INST
	fbCaseTest0203				: FB_CASE_ValidateContent;
	rTrig0203					: R_TRIG;
	nCycles0203					: INT;
	
END_VAR

//Data initialization
TestInit(stCACData:= stCACData_test_0203, stProductInstruction:= stProductInstruction_test_0203);

//Change some data for test scenario below
stCACData_test_0203.NumberOfOuters := - 2;
	
TcUnit.TEST('dataConsistancy03_ValidationCodeNotFoundInInfeedQueue');


fbCaseTest0203(
	bExecute:= TRUE, 
	bIsDuplicateOuters:= FALSE, 
	bIsDuplicatePacks:= FALSE, 
	stCTDateTime:= stCTDateTime_tests, 
	stOuterDataNotFound:= stRejectReasonsForOuter_tests.stOuterDataNotFound, 
	stProductInstruction:= stProductInstruction_test_0203, 
	nSecquentionalCounter:= nSecquentionalCounter_tests, 
	stCodeInfo_Outer:= stCodeInfo_Outer_tests, 
	stCaseRejectReasons:= stCaseRejectReasons_tests, 
	stCACData:= stCACData_test_0203, 
	bDone=> bDone, 
	bBusy=> bBusy, 
	bError=> bError, 
	nErrorID=> nErrorID, 
	sRejectCode=> sRejectCode_test_0203, 
	nValidationIndex=> nValidationIndex
);
	
rTrig0203(CLK:= fbCaseTest0203.bDone);
nCycles0203 := nCycles0203 + 1;	

IF rTrig0203.Q THEN	
		
	AssertEquals_UDINT(Expected := 12,
                   	   Actual 	:= fbCaseTest0203.nErrorID,
                   	   Message 	:= 'nErrorID value wrong');
	
	TEST_FINISHED();
	
ELSIF nCycles0203 > 50 THEN
	
	AssertTrue(Condition := TRUE,
			   Message 	 := 'Timeout dataConsistancy03_ValidationCodeNotFoundInInfeedQueue'
	);	 
	TEST_FINISHED();
END_IF
END_METHOD

METHOD INTERNAL dataConsistancy04_OuterCodeVal_IndexErrorFound
VAR
	//fbCaseTest			: FB_CASE_ValidateContent;
	bDone				: BOOL;
	bBusy				: BOOL;
	bError				: BOOL;
	nErrorID 			: UDINT;
	nValidationIndex	: INT;
	
	eLastState			: E_CAC_State;
			
END_VAR

VAR_INST
	fbCaseTest0204				: FB_CASE_ValidateContent;
	rTrig0204					: R_TRIG;
	nCycles0204					: INT;
	
END_VAR

//Data initialization
TestInit(stCACData:= stCACData_test_0204, stProductInstruction:= stProductInstruction_test_0204);

//Change some data for test scenario below
stCACData_test_0204.NumberOfOuters := - 3;
	
TcUnit.TEST('dataConsistancy04_OuterCodeVal_IndexErrorFound');


fbCaseTest0204(
	bExecute:= TRUE, 
	bIsDuplicateOuters:= FALSE, 
	bIsDuplicatePacks:= FALSE, 
	stCTDateTime:= stCTDateTime_tests, 
	stOuterDataNotFound:= stRejectReasonsForOuter_tests.stOuterDataNotFound, 
	stProductInstruction:= stProductInstruction_test_0204, 
	nSecquentionalCounter:= nSecquentionalCounter_tests, 
	stCodeInfo_Outer:= stCodeInfo_Outer_tests, 
	stCaseRejectReasons:= stCaseRejectReasons_tests, 
	stCACData:= stCACData_test_0204, 
	bDone=> bDone, 
	bBusy=> bBusy, 
	bError=> bError, 
	nErrorID=> nErrorID, 
	sRejectCode=> sRejectCode_test_0204, 
	nValidationIndex=> nValidationIndex
);
	
rTrig0204(CLK:= fbCaseTest0204.bDone);
nCycles0204 := nCycles0204 + 1;	

IF rTrig0204.Q THEN	
		
	AssertEquals_UDINT(Expected := 13,
                   	   Actual 	:= fbCaseTest0204.nErrorID,
                   	   Message 	:= 'nErrorID value wrong');
	
	TEST_FINISHED();
	
ELSIF nCycles0204 > 50 THEN
	
	AssertTrue(Condition := TRUE,
			   Message 	 := 'Timeout dataConsistancy04_OuterCodeVal_IndexErrorFound'
	);	 
	TEST_FINISHED();
END_IF
END_METHOD

METHOD INTERNAL dataConsistancy05_NumberOfOutersToSmall
VAR
	//fbCaseTest			: FB_CASE_ValidateContent;
	bDone				: BOOL;
	bBusy				: BOOL;
	bError				: BOOL;
	nErrorID 			: UDINT;
	nValidationIndex	: INT;
	
	eLastState			: E_CAC_State;
			
END_VAR

VAR_INST
	fbCaseTest0205				: FB_CASE_ValidateContent;
	rTrig0205					: R_TRIG;
	nCycles0205					: INT;
	
END_VAR

//Data initialization
TestInit(stCACData:= stCACData_test_0205, stProductInstruction:= stProductInstruction_test_0205);

//Change some data for test scenario below
stCACData_test_0205.NumberOfOuters := 25;
	
TcUnit.TEST('dataConsistancy05_NumberOfOutersToSmall');


fbCaseTest0205(
	bExecute:= TRUE, 
	bIsDuplicateOuters:= FALSE, 
	bIsDuplicatePacks:= FALSE, 
	stCTDateTime:= stCTDateTime_tests, 
	stOuterDataNotFound:= stRejectReasonsForOuter_tests.stOuterDataNotFound, 
	stProductInstruction:= stProductInstruction_test_0205, 
	nSecquentionalCounter:= nSecquentionalCounter_tests, 
	stCodeInfo_Outer:= stCodeInfo_Outer_tests, 
	stCaseRejectReasons:= stCaseRejectReasons_tests, 
	stCACData:= stCACData_test_0205, 
	bDone=> bDone, 
	bBusy=> bBusy, 
	bError=> bError, 
	nErrorID=> nErrorID, 
	sRejectCode=> sRejectCode_test_0205, 
	nValidationIndex=> nValidationIndex
);
	
rTrig0205(CLK:= fbCaseTest0205.bDone);
nCycles0205 := nCycles0205 + 1;	

IF rTrig0205.Q THEN	
		
	AssertEquals_UDINT(Expected := 14,
                   	   Actual 	:= fbCaseTest0205.nErrorID,
                   	   Message 	:= 'nErrorID value wrong');
	
	TEST_FINISHED();
	
ELSIF nCycles0205 > 50 THEN
	
	AssertTrue(Condition := TRUE,
			   Message 	 := 'Timeout dataConsistancy05_NumberOfOutersToSmall'
	);	 
	TEST_FINISHED();
END_IF
END_METHOD

METHOD INTERNAL dataConsistancy06_NumberOfOutersToBig
VAR
	//fbCaseTest			: FB_CASE_ValidateContent;
	bDone				: BOOL;
	bBusy				: BOOL;
	bError				: BOOL;
	nErrorID 			: UDINT;
	nValidationIndex	: INT;
	
	eLastState			: E_CAC_State;
			
END_VAR

VAR_INST
	fbCaseTest0206				: FB_CASE_ValidateContent;
	rTrig0206					: R_TRIG;
	nCycles0206					: INT;
	
END_VAR

//Data initialization
TestInit(stCACData:= stCACData_test_0206, stProductInstruction:= stProductInstruction_test_0206);

//Change some data for test scenario below
stCACData_test_0206.NumberOfOuters := 69;
	
TcUnit.TEST('dataConsistancy06_NumberOfOutersToBig');


fbCaseTest0206(
	bExecute:= TRUE, 
	bIsDuplicateOuters:= FALSE, 
	bIsDuplicatePacks:= FALSE, 
	stCTDateTime:= stCTDateTime_tests, 
	stOuterDataNotFound:= stRejectReasonsForOuter_tests.stOuterDataNotFound, 
	stProductInstruction:= stProductInstruction_test_0206, 
	nSecquentionalCounter:= nSecquentionalCounter_tests, 
	stCodeInfo_Outer:= stCodeInfo_Outer_tests, 
	stCaseRejectReasons:= stCaseRejectReasons_tests, 
	stCACData:= stCACData_test_0206, 
	bDone=> bDone, 
	bBusy=> bBusy, 
	bError=> bError, 
	nErrorID=> nErrorID, 
	sRejectCode=> sRejectCode_test_0206, 
	nValidationIndex=> nValidationIndex
);
	
rTrig0206(CLK:= fbCaseTest0206.bDone);
nCycles0206 := nCycles0206 + 1;	

IF rTrig0206.Q THEN	
		
	AssertEquals_UDINT(Expected := 15,
                   	   Actual 	:= fbCaseTest0206.nErrorID,
                   	   Message 	:= 'nErrorID value wrong');
	
	TEST_FINISHED();
	
ELSIF nCycles0206 > 50 THEN
	
	AssertTrue(Condition := TRUE,
			   Message 	 := 'Timeout dataConsistancy06_NumberOfOutersToBig'
	);	 
	TEST_FINISHED();
END_IF
END_METHOD

METHOD INTERNAL duplicateHandler01_OuterDuplicatebErrorTrue
VAR
	//fbCaseTest			: FB_CASE_ValidateContent;
	bDone				: BOOL;
	bBusy				: BOOL;
	bError				: BOOL;
	nErrorID 			: UDINT;
	nValidationIndex	: INT;
	
	eLastState			: E_CAC_State;
			
END_VAR

VAR_INST
	fbCaseTest0601				: FB_CASE_ValidateContent;
	fTrig						: F_TRIG;	
	rTrig						: R_TRIG;
	nCycles						: INT;
	
END_VAR

//Data initialization
TestInit(stCACData:= stCACData_test_0601, stProductInstruction:= stProductInstruction_test_0601);

//Change some data for test scenario below
//stCACData_test_0303.NumberOfOuters := 51;

	
TcUnit.TEST('duplicateHandler01_OuterDuplicatebErrorTrue');


fbCaseTest0601(
	bExecute:= TRUE, 
	bIsDuplicateOuters:= TRUE, 
	bIsDuplicatePacks:= FALSE, 
	stCTDateTime:= stCTDateTime_tests, 
	stOuterDataNotFound:= stRejectReasonsForOuter_tests.stOuterDataNotFound, 
	stProductInstruction:= stProductInstruction_test_0601, 
	nSecquentionalCounter:= nSecquentionalCounter_tests, 
	stCodeInfo_Outer:= stCodeInfo_Outer_tests, 
	stCaseRejectReasons:= stCaseRejectReasons_tests, 
	stCACData:= stCACData_test_0601, 
	bDone=> bDone, 
	bBusy=> bBusy, 
	bError=> bError, 
	nErrorID=> nErrorID, 
	sRejectCode=> sRejectCode_tets, 
	nValidationIndex=> nValidationIndex
);
	
rTrig(CLK:= fbCaseTest0601.bDone);
nCycles := nCycles + 1;	

IF rTrig.Q THEN	
		
	AssertEquals_BOOL(Expected 	:= TRUE,
					  Actual 	:= bError,
					  Message 	:= 'Outer duplicate did not call error'
	);
	
	AssertEquals_UDINT(Expected := 1,
                   	   Actual 	:= fbCaseTest0601.nErrorID,
                   	   Message 	:= 'Wrong nErrorID on outer duplicate'
	);
	
	TEST_FINISHED();
	
ELSIF nCycles > 50 THEN
	
	AssertTrue(Condition := TRUE,
			   Message 	 := 'Timeout duplicateHandler01_OuterDuplicatebErrorTrue'
	);	 
	TEST_FINISHED();
END_IF
END_METHOD

METHOD INTERNAL duplicateHandler02_PackDuplicatebErrorTrue
VAR
	//fbCaseTest			: FB_CASE_ValidateContent;
	bDone				: BOOL;
	bBusy				: BOOL;
	bError				: BOOL;
	nErrorID 			: UDINT;
	nValidationIndex	: INT;
	
	eLastState			: E_CAC_State;
			
END_VAR

VAR_INST
	fbCaseTest0602				: FB_CASE_ValidateContent;
	fTrig						: F_TRIG;	
	rTrig						: R_TRIG;
	nCycles						: INT;
	
END_VAR

//Data initialization
TestInit(stCACData:= stCACData_test_0602, stProductInstruction:= stProductInstruction_test_0602);

//Change some data for test scenario below

	
TcUnit.TEST('duplicateHandler02_PackDuplicatebErrorTrue');


fbCaseTest0602(
	bExecute:= TRUE, 
	bIsDuplicateOuters:= FALSE, 
	bIsDuplicatePacks:= TRUE, 
	stCTDateTime:= stCTDateTime_tests, 
	stOuterDataNotFound:= stRejectReasonsForOuter_tests.stOuterDataNotFound, 
	stProductInstruction:= stProductInstruction_test_0602, 
	nSecquentionalCounter:= nSecquentionalCounter_tests, 
	stCodeInfo_Outer:= stCodeInfo_Outer_tests, 
	stCaseRejectReasons:= stCaseRejectReasons_tests, 
	stCACData:= stCACData_test_0602, 
	bDone=> bDone, 
	bBusy=> bBusy, 
	bError=> bError, 
	nErrorID=> nErrorID, 
	sRejectCode=> sRejectCode_tets, 
	nValidationIndex=> nValidationIndex
);
	
rTrig(CLK:= fbCaseTest0602.bDone);
nCycles := nCycles + 1;	

IF rTrig.Q THEN	
		
	AssertEquals_BOOL(Expected 	:= TRUE,
					  Actual 	:= bError,
					  Message 	:= 'Pack duplicate did not call error'
	);
	
	AssertEquals_UDINT(Expected := 1,
                   	   Actual 	:= fbCaseTest0602.nErrorID,
                   	   Message 	:= 'Wrong nErrorID on pack duplicate'
	);
	
	TEST_FINISHED();
	
ELSIF nCycles > 50 THEN
	
	AssertTrue(Condition := TRUE,
			   Message 	 := 'Timeout duplicateHandler02_PackDuplicatebErrorTrue'
	);	 
	TEST_FINISHED();
END_IF
END_METHOD

METHOD INTERNAL main01_bExecuteFalseNoAction
VAR
	//fbCaseTest			: FB_CASE_ValidateContent;
	bDone				: BOOL;
	bBusy				: BOOL;
	bError				: BOOL;
	nErrorID 			: UDINT;
	nValidationIndex	: INT;
	
	eLastState			: E_CAC_State;
			
END_VAR

VAR_INST
	fbCaseTest0101				: FB_CASE_ValidateContent;
	fTrig						: F_TRIG;	
	rTrig						: R_TRIG;
	nCycles						: INT;
	
END_VAR

//Data initialization
TestInit(stCACData:= stCACData_test_0101, stProductInstruction:= stProductInstruction_test_0101);

//Change some data for test scenario below

	
TcUnit.TEST('main01_bExecuteFalseNoAction');


fbCaseTest0101(
	bExecute:= FALSE, 
	bIsDuplicateOuters:= FALSE, 
	bIsDuplicatePacks:= FALSE, 
	stCTDateTime:= stCTDateTime_tests, 
	stOuterDataNotFound:= stRejectReasonsForOuter_tests.stOuterDataNotFound, 
	stProductInstruction:= stProductInstruction_test_0101, 
	nSecquentionalCounter:= nSecquentionalCounter_tests, 
	stCodeInfo_Outer:= stCodeInfo_Outer_tests, 
	stCaseRejectReasons:= stCaseRejectReasons_tests, 
	stCACData:= stCACData_test_0101, 
	bDone=> bDone, 
	bBusy=> bBusy, 
	bError=> bError, 
	nErrorID=> nErrorID, 
	sRejectCode=> sRejectCode_tets, 
	nValidationIndex=> nValidationIndex
);
	
rTrig(CLK:= fbCaseTest0101.bDone);
nCycles := nCycles + 1;	

		
AssertEquals_BOOL(Expected 	:= FALSE,
				  Actual 	:= fbCaseTest0101.bError,
				  Message 	:= 'FB no executed wrong output'
);

AssertEquals_BOOL(Expected 	:= FALSE,
				  Actual 	:= fbCaseTest0101.bDone,
				  Message 	:= 'B no executed wrong output'
);

TEST_FINISHED();
END_METHOD

METHOD INTERNAL numberOfOuters01_ValueToLittlebErrorTrue
VAR
	//fbCaseTest			: FB_CASE_ValidateContent;
	bDone				: BOOL;
	bBusy				: BOOL;
	bError				: BOOL;
	nErrorID 			: UDINT;
	nValidationIndex	: INT;
	
	eLastState			: E_CAC_State;
			
END_VAR

VAR_INST
	fbCaseTest0301				: FB_CASE_ValidateContent;
	fTrig0301						: F_TRIG;
	nCycles0301						: INT;
	
END_VAR

//Data initialization
TestInit(stCACData:= stCACData_test_0301, stProductInstruction:= stProductInstruction_test_0301);

//Change some data for test scenario below
stCACData_test_0301.NumberOfOuters := 45;
	


TcUnit.TEST('numberOfOuters01_ValueToLittlebErrorTrue');

fbCaseTest0301(
	bExecute:= TRUE, 
	bIsDuplicateOuters:= FALSE, 
	bIsDuplicatePacks:= FALSE, 
	stCTDateTime:= stCTDateTime_tests, 
	stOuterDataNotFound:= stRejectReasonsForOuter_tests.stOuterDataNotFound, 
	stProductInstruction:= stProductInstruction_test_0301, 
	nSecquentionalCounter:= nSecquentionalCounter_tests, 
	stCodeInfo_Outer:= stCodeInfo_Outer_tests, 
	stCaseRejectReasons:= stCaseRejectReasons_tests, 
	stCACData:= stCACData_test_0301, 
	bDone=> bDone, 
	bBusy=> bBusy, 
	bError=> bError, 
	nErrorID=> nErrorID, 
	sRejectCode=> sRejectCode_test_0301, 
	nValidationIndex=> nValidationIndex
);

fTrig0301(CLK:= fbCaseTest0301.bBusy);
nCycles0301 := nCycles0301 + 1;	

IF fTrig0301.Q AND nCycles0301 <= 50 THEN	
	
	AssertEquals_BOOL(Expected := TRUE,
					  Actual := fbCaseTest0301.bError,
					  Message := 'Numbers of outer wrong value didnt call error'
	);
	
	AssertEquals_STRING(Expected := 'XXVAL045XX',
						Actual := TO_STRING(fbCaseTest0301.sRejectCode),
						Message := 'Wrong value of nErrorID'
	);
	
	AssertEquals_INT(Expected := 45,
					 Actual := stCACData_test_0301.NumberOfOuters,
					 Message := 'INT Values differ'
	);	
	
	TEST_FINISHED();
	
ELSIF nCycles0301 > 50 THEN
	
	AssertTrue(Condition := TRUE,
			   Message := 'Timeout CASE loop within FB_CASE_Validation'
	);	 

	
	TEST_FINISHED();
END_IF
END_METHOD

METHOD INTERNAL numberOfOuters02_ValueGraterErrorTrue
VAR
	
	bDone				: BOOL;
	bBusy				: BOOL;
	bError				: BOOL;
	nErrorID 			: UDINT;
	nValidationIndex	: INT;
	
	eLastState			: E_CAC_State;
	
		
END_VAR

VAR_INST
	
	fbCaseTest0302				: FB_CASE_ValidateContent;
	fTrig0302						: F_TRIG;
	nCycles0302						: INT;
	
END_VAR

//Data initialization
TestInit(stCACData:= stCACData_test_0302, stProductInstruction:= stProductInstruction_test_0302);

//Change some data for test scenario below
stCACData_test_0302.NumberOfOuters := 79;

	
TcUnit.TEST('numberOfOuters02_ValueGraterErrorTrue');


fbCaseTest0302(
	bExecute:= TRUE, 
	bIsDuplicateOuters:= FALSE, 
	bIsDuplicatePacks:= FALSE, 
	stCTDateTime:= stCTDateTime_tests, 
	stOuterDataNotFound:= stRejectReasonsForOuter_tests.stOuterDataNotFound, 
	stProductInstruction:= stProductInstruction_test_0302, 
	nSecquentionalCounter:= nSecquentionalCounter_tests, 
	stCodeInfo_Outer:= stCodeInfo_Outer_tests, 
	stCaseRejectReasons:= stCaseRejectReasons_tests, 
	stCACData:= stCACData_test_0302, 
	bDone=> bDone, 
	bBusy=> bBusy, 
	bError=> bError, 
	nErrorID=> nErrorID, 
	sRejectCode=> sRejectCode_test_0302, 
	nValidationIndex=> nValidationIndex
);
	
fTrig0302(CLK:= fbCaseTest0302.bBusy);
nCycles0302 := nCycles0302 + 1;	

IF fTrig0302.Q AND nCycles0302 <= 50 THEN	
		
	AssertEquals_BOOL(Expected := TRUE,
					  Actual := fbCaseTest0302.bError,
					  Message := 'Numbers of outer wrong value didnt call error'
	);
	
	AssertEquals_STRING(Expected := 'XXVAL079XX',
						Actual := TO_STRING(fbCaseTest0302.sRejectCode),
						Message := 'Wrong value of sRejectCode'
	);
	
	TEST_FINISHED();
	
ELSIF nCycles0302 > 50 THEN
	
	AssertTrue(Condition := TRUE,
			   Message 	 := 'Timeout numberOfOuters02_ValueGraterErrorTrue'
	);	 
	
	TEST_FINISHED();
END_IF
END_METHOD

METHOD INTERNAL numberOfOuters03_ValueToLittlebErrorTrueRejectCodeWright
VAR
	//fbCaseTest			: FB_CASE_ValidateContent;
	bDone				: BOOL;
	bBusy				: BOOL;
	bError				: BOOL;
	nErrorID 			: UDINT;
	nValidationIndex	: INT;
	
	eLastState			: E_CAC_State;
			
END_VAR

VAR_INST
	fbCaseTest0303				: FB_CASE_ValidateContent;
	fTrig						: F_TRIG;
	nCycles						: INT;
	
END_VAR

//Data initialization
TestInit(stCACData:= stCACData_test_0303, stProductInstruction:= stProductInstruction_test_0303);

//Change some data for test scenario below
stCACData_test_0303.NumberOfOuters := 51;

	
TcUnit.TEST('numberOfOuters03_ValueToLittlebErrorTrueRejectCodeWright');


fbCaseTest0303(
	bExecute:= TRUE, 
	bIsDuplicateOuters:= FALSE, 
	bIsDuplicatePacks:= FALSE, 
	stCTDateTime:= stCTDateTime_tests, 
	stOuterDataNotFound:= stRejectReasonsForOuter_tests.stOuterDataNotFound, 
	stProductInstruction:= stProductInstruction_test_0301, 
	nSecquentionalCounter:= nSecquentionalCounter_tests, 
	stCodeInfo_Outer:= stCodeInfo_Outer_tests, 
	stCaseRejectReasons:= stCaseRejectReasons_tests, 
	stCACData:= stCACData_test_0303, 
	bDone=> bDone, 
	bBusy=> bBusy, 
	bError=> bError, 
	nErrorID=> nErrorID, 
	sRejectCode=> sRejectCode_test_0303, 
	nValidationIndex=> nValidationIndex
);
	
fTrig(CLK:= fbCaseTest0303.bBusy);
nCycles := nCycles + 1;	

IF fTrig.Q THEN	
		
	AssertEquals_BOOL(Expected := TRUE,
					  Actual := fbCaseTest0303.bError,
					  Message := 'Numbers of outer wrong value didnt call error'
	);
	
	AssertEquals_STRING(Expected := 'XXVAL051XX',
						Actual := TO_STRING(fbCaseTest0303.sRejectCode),
						Message := 'Wrong value of sRejectCode'
	);
	
	TEST_FINISHED();
	
ELSIF nCycles > 50 THEN
	
	AssertTrue(Condition := TRUE,
			   Message 	 := 'Timeout numberOfOuters03_ValueToLittlebErrorTrueRejectCodeWright'
	);	 
	
	TEST_FINISHED();
END_IF
END_METHOD

METHOD INTERNAL oacMissing01nErrorID21
VAR
	//fbCaseTest			: FB_CASE_ValidateContent;
	bDone				: BOOL;
	bBusy				: BOOL;
	bError				: BOOL;
	nErrorID 			: UDINT;
	nValidationIndex	: INT;
	bCompare			: BOOL;
	
	eLastState			: E_CAC_State;
			
END_VAR

VAR_INST
	fbCaseTest0701				: FB_CASE_ValidateContent;
	fTrig0701					: F_TRIG;	
	rTrig0701					: R_TRIG;
	nCycles0701					: INT;
	
END_VAR

//Data initialization
TestInit(stCACData:= stCACData_test_0701, stProductInstruction:= stProductInstruction_test_0701);

//Change some data for test scenario below
stCACData_test_0701.Outer[5].OuterRejectID := 207;
stProductInstruction_test_0701.nCaseAcceptanceLevelOuters := 50;
	
TcUnit.TEST('oacMissing01nErrorID21');


fbCaseTest0701(
	bExecute:= TRUE, 
	bIsDuplicateOuters:= FALSE, 
	bIsDuplicatePacks:= FALSE, 
	stCTDateTime:= stCTDateTime_tests, 
	stOuterDataNotFound:= stRejectReasonsForOuter_tests.stOuterDataNotFound, 
	stProductInstruction:= stProductInstruction_test_0701, 
	nSecquentionalCounter:= nSecquentionalCounter_tests, 
	stCodeInfo_Outer:= stCodeInfo_Outer_tests, 
	stCaseRejectReasons:= stCaseRejectReasons_tests, 
	stCACData:= stCACData_test_0701, 
	bDone=> bDone, 
	bBusy=> bBusy, 
	bError=> bError, 
	nErrorID=> nErrorID, 
	sRejectCode=> sRejectCode_tets, 
	nValidationIndex=> nValidationIndex
);
	
rTrig0701(CLK:= fbCaseTest0701.bDone);
nCycles0701 := nCycles0701 + 1;	



IF rTrig0701.Q THEN	
	
	bCompare := (stCACData_test_0701.CaseRejectID = stCaseRejectReasons_tests.stOACError.nRejectID);
	
	AssertEquals_BOOL(Expected 	:= TRUE,
					  Actual 	:= bError,
					  Message 	:= 'Pack duplicate did not call error'
	);
	
	AssertEquals_UDINT(Expected := 21,
                   	   Actual 	:= fbCaseTest0701.nErrorID,
                   	   Message 	:= 'Wrong nErrorID on OAC missing'
	);
	
	AssertEquals_BOOL(Expected 	:= TRUE,
					  Actual 	:= bCompare,
					  Message 	:= 'CaseRejectID wrong value'
	);	
	
	TEST_FINISHED();
	
ELSIF nCycles0701 > 50 THEN
	
	AssertTrue(Condition := TRUE,
			   Message 	 := 'Timeout oacMissing01nErrorID21'
	);	 
	TEST_FINISHED();
END_IF
END_METHOD

METHOD INTERNAL outerAggrDissable01_sRejectCodeOK
VAR
	//fbCaseTest			: FB_CASE_ValidateContent;
	bDone				: BOOL;
	bBusy				: BOOL;
	bError				: BOOL;
	nErrorID 			: UDINT;
	nValidationIndex	: INT;
	
	eLastState			: E_CAC_State;
			
END_VAR

VAR_INST
	fbCaseTest0401				: FB_CASE_ValidateContent;
	rTrig0401					: R_TRIG;
	nCycles0401					: INT;
	
END_VAR

//Data initialization
TestInit(stCACData:= stCACData_test_0401, stProductInstruction:= stProductInstruction_test_0401);

//Change some data for test scenario below
stCACData_test_0401.CodingAndTrackingMode := 6;
	
TcUnit.TEST('outerAggrDissable01_sRejectCodeOK');


fbCaseTest0401(
	bExecute:= TRUE, 
	bIsDuplicateOuters:= FALSE, 
	bIsDuplicatePacks:= FALSE, 
	stCTDateTime:= stCTDateTime_tests, 
	stOuterDataNotFound:= stOuterDataNotFound_tests, 
	stProductInstruction:= stProductInstruction_test_0401, 
	nSecquentionalCounter:= nSecquentionalCounter_tests, 
	stCodeInfo_Outer:= stCodeInfo_Outer_tests, 
	stCaseRejectReasons:= stCaseRejectReasons_tests, 
	stCACData:= stCACData_test_0401, 
	bDone=> bDone, 
	bBusy=> bBusy, 
	bError=> bError, 
	nErrorID=> nErrorID, 
	sRejectCode=> sRejectCode_test_0401, 
	nValidationIndex=> nValidationIndex
);
	
rTrig0401(CLK:= fbCaseTest0401.bDone);
nCycles0401 := nCycles0401 + 1;	

IF rTrig0401.Q THEN	
	
	AssertEquals_STRING(Expected := 'OK',
						Actual := TO_STRING(fbCaseTest0401.sRejectCode),
						Message := 'Wrong value of nErrorID'
	);
	
	
	TEST_FINISHED();
	
ELSIF nCycles0401 > 50 THEN
	
	AssertTrue(Condition := TRUE,
			   Message 	 := 'Timeout outerAggrDissable01_sRejectCodeOK'
	);	 
	TEST_FINISHED();
END_IF
END_METHOD

METHOD INTERNAL outerAggrEnable01_PacksPerOuterZero
VAR
	//fbCaseTest			: FB_CASE_ValidateContent;
	bDone				: BOOL;
	bBusy				: BOOL;
	bError				: BOOL;
	nErrorID 			: UDINT;
	nValidationIndex	: INT;
	
	eLastState			: E_CAC_State;
			
END_VAR

VAR_INST
	fbCaseTest0501				: FB_CASE_ValidateContent;
	rTrig0501					: R_TRIG;
	nCycles0501					: INT;
	
END_VAR

//Data initialization
TestInit(stCACData:= stCACData_test_0501, stProductInstruction:= stProductInstruction_test_0501);

//Change some data for test scenario below
stCACData_test_0501.CodingAndTrackingMode := 8;
stProductInstruction_test_0501.nPacksPerOuter := 0;
	
TcUnit.TEST('outerAggrEnable01_PacksPerOuterZero');


fbCaseTest0501(
	bExecute:= TRUE, 
	bIsDuplicateOuters:= FALSE, 
	bIsDuplicatePacks:= FALSE, 
	stCTDateTime:= stCTDateTime_tests, 
	stOuterDataNotFound:= stRejectReasonsForOuter_tests.stOuterDataNotFound, 
	stProductInstruction:= stProductInstruction_test_0501, 
	nSecquentionalCounter:= nSecquentionalCounter_tests, 
	stCodeInfo_Outer:= stCodeInfo_Outer_tests, 
	stCaseRejectReasons:= stCaseRejectReasons_tests, 
	stCACData:= stCACData_test_0501, 
	bDone=> bDone, 
	bBusy=> bBusy, 
	bError=> bError, 
	nErrorID=> nErrorID, 
	sRejectCode=> sRejectCode_test_0501, 
	nValidationIndex=> nValidationIndex
);
	
rTrig0501(CLK:= fbCaseTest0501.bDone);
nCycles0501 := nCycles0501 + 1;	

IF rTrig0501.Q THEN	
	
	AssertEquals_BOOL(Expected 	:= TRUE,
					  Actual 	:= bError,
					  Message 	:= 'Wrong number of outers not detected'
	);

	AssertEquals_UDINT(Expected := 10,
                   	   Actual 	:= fbCaseTest0501.nErrorID,
                   	   Message 	:= 'nErrorID value wrong'
	);
	
	
	TEST_FINISHED();
	
ELSIF nCycles0501 > 50 THEN
	
	AssertTrue(Condition := TRUE,
			   Message 	 := 'Timeout outerAggrEnable01_PacksPerOuterZero'
	);	 
	TEST_FINISHED();
END_IF
END_METHOD

METHOD INTERNAL outerAggrEnable02_PacksPerCaseZero
VAR
	//fbCaseTest			: FB_CASE_ValidateContent;
	bDone				: BOOL;
	bBusy				: BOOL;
	bError				: BOOL;
	nErrorID 			: UDINT;
	nValidationIndex	: INT;
	
	eLastState			: E_CAC_State;
			
END_VAR

VAR_INST
	fbCaseTest0502				: FB_CASE_ValidateContent;
	rTrig0502					: R_TRIG;
	nCycles0502					: INT;
	
END_VAR

//Data initialization
TestInit(stCACData:= stCACData_test_0502, stProductInstruction:= stProductInstruction_test_0502);

//Change some data for test scenario below
stCACData_test_0502.CodingAndTrackingMode := 8;
stProductInstruction_test_0502.nPacksPerCase := 0;
	
TcUnit.TEST('outerAggrEnable02_PacksPerCaseZero');


fbCaseTest0502(
	bExecute:= TRUE, 
	bIsDuplicateOuters:= FALSE, 
	bIsDuplicatePacks:= FALSE, 
	stCTDateTime:= stCTDateTime_tests, 
	stOuterDataNotFound:= stRejectReasonsForOuter_tests.stOuterDataNotFound, 
	stProductInstruction:= stProductInstruction_test_0502, 
	nSecquentionalCounter:= nSecquentionalCounter_tests, 
	stCodeInfo_Outer:= stCodeInfo_Outer_tests, 
	stCaseRejectReasons:= stCaseRejectReasons_tests, 
	stCACData:= stCACData_test_0502, 
	bDone=> bDone, 
	bBusy=> bBusy, 
	bError=> bError, 
	nErrorID=> nErrorID, 
	sRejectCode=> sRejectCode_test_0502, 
	nValidationIndex=> nValidationIndex
);
	
rTrig0502(CLK:= fbCaseTest0502.bDone);
nCycles0502 := nCycles0502 + 1;	

IF rTrig0502.Q THEN	
	
	AssertEquals_BOOL(Expected 	:= TRUE,
					  Actual 	:= bError,
					  Message 	:= 'Wrong number of outers not detected'
	);

	AssertEquals_UDINT(Expected := 10,
                   	   Actual 	:= fbCaseTest0502.nErrorID,
                   	   Message 	:= 'nErrorID value wrong'
	);
	
	
	TEST_FINISHED();
	
ELSIF nCycles0502 > 50 THEN
	
	AssertTrue(Condition := TRUE,
			   Message 	 := 'Timeout outerAggrEnable02_PacksPerCaseZero'
	);	 
	TEST_FINISHED();
END_IF
END_METHOD

METHOD PRIVATE TestInit : BOOL
VAR_IN_OUT
	stProductInstruction	: ST_PCM_Status;
	stCACData 				: ST_CAC_Data;
END_VAR

VAR	
	rTrigDataInit		: R_TRIG;
	bDataInit			: BOOL;
	iOuter				: INT;
	iPack				: INT;
	sPackNum			: STRING;
	sOuterNum			: STRING;
	sPackCode			: STRING;
END_VAR

VAR_OUTPUT
	bDone				: BOOL;
END_VAR

//MEMSET(ADR(stCACData), 16#00, SIZEOF(stCACData));	

stProductInstruction.nOutersPerCase 	:= 50;
stProductInstruction.nPacksPerOuter		:= 10;
stProductInstruction.nPacksPerCase		:= 500;
stProductInstruction.nOpMode			:= 11;
stProductInstruction.sRetailSKU			:= '1234567';
stProductInstruction.nAcceptanceLevel 	:= 10;

stCACData.NumberOfOuters			:= stProductInstruction.nOutersPerCase;
stCACData.CodingAndTrackingMode		:= stProductInstruction.nOpMode;
stCACData.RetailSKU					:= stProductInstruction.sRetailSKU;

FOR iOuter := 1 TO stProductInstruction.nOutersPerCase DO
	(* Outer number z zerami *)
	sOuterNum := F_StringAddPrefix(INT_TO_STRING(iOuter),2,'0');

	stCACData.Outer[iOuter].Barcode    				:= CONCAT('OUTER', sOuterNum);
	stCACData.Outer[iOuter].NumberOfPacks 			:= stProductInstruction.nPacksPerOuter;
	stCACData.Outer[iOuter].NumberOfLinkedPacks 	:= stProductInstruction.nPacksPerOuter;
	stCACData.Outer[iOuter].AcceptanceLevel 		:= stProductInstruction.nAcceptanceLevel;
	stCACData.Outer[iOuter].CodingAndTrackingMode	:= stProductInstruction.nOpMode;
	stCACData.Outer[iOuter].OuterRejectCode			:= 'OK';

	FOR iPack := 1 TO stProductInstruction.nPacksPerOuter DO
		(* Pack number dwucyfrowy z zerami *)
		sPackNum := F_StringAddPrefix(INT_TO_STRING(iPack),2,'0');			
		(* Sklej pack code *)
		sPackCode := CONCAT(CONCAT('PACK', sPackNum), CONCAT('OUTER', sOuterNum));
		
		(* Write Pack Barcodes / Data*)
		stCACData.Outer[iOuter].PackCode[iPack]				:= sPackCode;
		stCACData.Outer[iOuter].PackCodeStatus[iPack]		:= 5;
		stCACData.Outer[iOuter].PackRejectID[iPack]			:= 0;			
		stCACData.Outer[iOuter].PackRejectCode[iPack]		:= 'OK';			
		stCACData.Outer[iOuter].PackCodeStatus[iPack].5 	:= TRUE;
		
		
		IF iPack = 1 THEN
			stCACData.Outer[iOuter].AggregationCodes[1]	:= stCACData.Outer[iOuter].PackCode[iPack];
		END_IF
		IF iPack = 2 THEN
			stCACData.Outer[iOuter].AggregationCodes[2]	:= stCACData.Outer[iOuter].PackCode[iPack];
		END_IF
	END_FOR
END_FOR	

stCACData.Outer[3].OuterCodeStatus.5 	:= TRUE;
stCACData.Outer[4].OuterCodeStatus.5	:= TRUE;
END_METHOD

END_FUNCTION_BLOCK

// ---- POUs/METS/Common LIB/08_SOFTWARE LIB/String FBs/F_StringAddPrefix.TcPOU
(* add specified char(s) in front of a string to make up to specified length *)
FUNCTION F_StringAddPrefix : T_MaxString
VAR_INPUT
	sString		: T_MaxString;	(* initial string *)
	nTargetLen 		: UINT;			(* string length required *)
	sChar			: STRING(1);	(* char to be appended to string *)
END_VAR
VAR
	nStringLen		: UINT;
	nCharsReq		: uINT;
END_VAR
(*
-------------------------------------------------------------------------------------------------
Date		Version	Author	Comments
-------------------------------------------------------------------------------------------------
30/01/2015	3.00.00	PB		Initial release

-------------------------------------------------------------------------------------------------
*)

(* length of input string *)
nStringLen := TO_UINT(LEN(sString));

(* Chekck target string is longer than processing string *)
IF nTargetLen >= nStringLen THEN
	
	(* total prefix chars required *)
	nCharsReq := MIN(nTargetLen, SIZEOF(F_StringAddPrefix) - 1) - nStringLen;

	(* string needs additional chars *)
	IF nCharsReq > 0 THEN
	
		(* set prefix chars to specified character *)
		MEMSET(ADR(F_StringAddPrefix), F_ToASC(sChar), nCharsReq);
	
		(* append strString to output string *)
		MEMMOVE(ADR(F_StringAddPrefix) + nCharsReq, ADR(sString), nStringLen);
	
		(* reset last char to 16#00 to terminate the string *)
		MEMSET(ADR(F_StringAddPrefix) + nCharsReq + nStringLen, 16#00, 1);
	
	(* no additional chars required *)
	ELSE
	
		(* copy strString to output *)
		F_StringAddPrefix := sString;
	END_IF
ELSE
	(* copy shrinced strString to output *)
	F_StringAddPrefix := LEFT(sString, TO_INT(nTargetLen));
END_IF

END_FUNCTION

// ---- POUs/TcUnit/FB_ExtractAnyStringTests/PRG_ExtractAnyStringManual.TcPOU
PROGRAM PRG_ExtractAnyStringManual
VAR
	fbExtractAnyString		: FB_ExtractAnyString;
	
	bExtractData		: BOOL;			(* set TRUE to remove prefix and suffix from strData *)
	nExtractChars		: UINT;			(* if suffix is blank, number of data chars to extract *)
	sPrefix				: T_MaxString;	(* prefix string *)
	sSuffix				: T_MaxString;	(* suffix string *)
	bIgnoreCase			: BOOL;
	eExtractMode		: E_STRING_ExtrMode	:= E_STRING_ExtrMode.WITHOUTIDENT_PURGE;

	sDataString			: T_LongSTRING;	(* string to be searched *)

	bStringFound				: BOOL;			(* TRUE = sub-string with matching prefix/suffix found *)
	sExtractedString			: T_LongSTRING;	(* extracted data *)
	nExtractedStringPos			: UDINT;			(* start pos of extracted string in strString *)
	nExtractedStringLen			: UDINT;
	nDataStringLen				: UDINT;
END_VAR

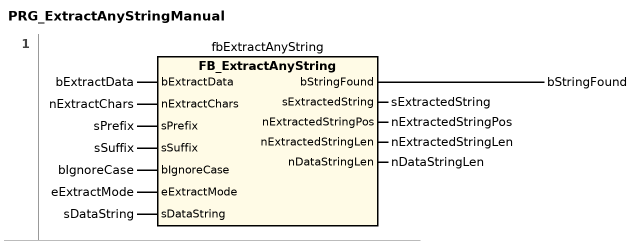
// NETWORK 1
fbExtractAnyString(
    bExtractData := bExtractData,
    nExtractChars := nExtractChars,
    sPrefix := sPrefix,
    sSuffix := sSuffix,
    bIgnoreCase := bIgnoreCase,
    eExtractMode := eExtractMode,
    sDataString := sDataString,
    sExtractedString => sExtractedString,
    nExtractedStringPos => nExtractedStringPos,
    nExtractedStringLen => nExtractedStringLen,
    nDataStringLen => nDataStringLen); // FB_ExtractAnyString
bStringFound := fbExtractAnyString.bStringFound;

END_PROGRAM

// ---- POUs/TcUnit/FB_ExtractStringTests/PRG_ExtractStringManual.TcPOU
PROGRAM PRG_ExtractStringManual
VAR
	fbExtractString		: FB_ExtractString;
	
	bExtractData		: BOOL;			(* set TRUE to remove prefix and suffix from strData *)
	nExtractChars		: UINT;			(* if suffix is blank, number of data chars to extract *)
	sPrefix				: T_MaxString;	(* prefix string *)
	sSuffix				: T_MaxString;	(* suffix string *)


	sDataString			: T_MaxString;	(* string to be searched *)

	bStringFound				: BOOL;			(* TRUE = sub-string with matching prefix/suffix found *)
	sExtractedString			: T_MaxString;	(* extracted data *)
	nExtractedStringPos			: UDINT;			(* start pos of extracted string in strString *)

	sResultString			: T_MaxString;	(* extracted data *)
END_VAR

